LIN {X -0.022,Y -255.168,Z 987.708,A 0.000,B 0.000,C 90.000,E1 307.443} C_DIS
LIN {X -0.119,Y -266.430,Z 987.696,A 0.000,B 0.000,C 90.000,E1 305.311} C_DIS
LIN {X 0.015,Y -280.721,Z 987.682,A 0.000,B 0.000,C 90.000,E1 302.832} C_DIS
LIN {X -0.071,Y -295.961,Z 987.669,A 0.000,B 0.000,C 90.000,E1 300.463} C_DIS
LIN {X 0.194,Y -314.730,Z 987.654,A 0.000,B 0.000,C 90.000,E1 297.769} C_DIS
LIN {X -0.075,Y -330.365,Z 987.644,A 0.000,B 0.000,C 90.000,E1 295.899} C_DIS
LIN {X -0.054,Y -352.007,Z 987.631,A 0.000,B 0.000,C 90.000,E1 293.567} C_DIS
LIN {X 0.003,Y -370.661,Z 987.621,A 0.000,B 0.000,C 90.000,E1 291.716} C_DIS
LIN {X -0.030,Y -387.055,Z 987.612,A 0.000,B 0.000,C 90.000,E1 290.174} C_DIS
LIN {X 0.079,Y -397.816,Z 987.606,A 0.000,B 0.000,C 90.000,E1 289.141} C_DIS
LIN {X 0.039,Y -408.356,Z 987.601,A 0.000,B 0.000,C 90.000,E1 288.127} C_DIS
LIN {X -0.163,Y -415.784,Z 987.597,A 0.000,B 0.000,C 90.000,E1 287.402} C_DIS
LIN {X 0.003,Y -425.654,Z 987.591,A 0.000,B 0.000,C 90.000,E1 286.315} C_DIS
LIN {X -0.019,Y -435.159,Z 987.585,A 0.000,B 0.000,C 90.000,E1 285.245} C_DIS
LIN {X 0.027,Y -444.217,Z 987.579,A 0.000,B 0.000,C 90.000,E1 284.175} C_DIS
LIN {X 0.074,Y -452.686,Z 987.573,A 0.000,B 0.000,C 90.000,E1 283.119} C_DIS
LIN {X -0.041,Y -458.562,Z 987.569,A 0.000,B 0.000,C 90.000,E1 282.355} C_DIS
LIN {X 0.178,Y -465.822,Z 987.563,A 0.000,B 0.000,C 90.000,E1 281.299} C_DIS
LIN {X 0.080,Y -470.862,Z 987.559,A 0.000,B 0.000,C 90.000,E1 280.546} C_DIS
LIN {X 0.034,Y -475.472,Z 987.554,A 0.000,B 0.000,C 90.000,E1 279.792} C_DIS
LIN {X 0.101,Y -479.412,Z 987.550,A 0.000,B 0.000,C 90.000,E1 279.029} C_DIS
LIN {X 0.128,Y -482.743,Z 987.546,A 0.000,B 0.000,C 90.000,E1 278.276} C_DIS
LIN {X 0.117,Y -485.467,Z 987.542,A 0.000,B 0.000,C 90.000,E1 277.530} C_DIS
LIN {X -0.179,Y -486.911,Z 987.539,A 0.000,B 0.000,C 90.000,E1 277.068} C_DIS
LIN {X 0.019,Y -488.089,Z 987.536,A 0.000,B 0.000,C 90.000,E1 276.549} C_DIS
LIN {X -0.260,Y -489.035,Z 987.534,A 0.000,B 0.000,C 90.000,E1 276.087} C_DIS
LIN {X -0.046,Y -489.695,Z 987.531,A 0.000,B 0.000,C 90.000,E1 275.568} C_DIS
LIN {X 0.171,Y -489.938,Z 987.528,A 0.000,B 0.000,C 90.000,E1 275.049} C_DIS
LIN {X -0.097,Y -489.761,Z 987.525,A 0.000,B 0.000,C 90.000,E1 274.588} C_DIS
LIN {X 0.086,Y -489.164,Z 987.523,A 0.000,B 0.000,C 90.000,E1 274.073} C_DIS
LIN {X -0.183,Y -488.056,Z 987.520,A 0.000,B 0.000,C 90.000,E1 273.612} C_DIS
LIN {X 0.027,Y -486.383,Z 987.517,A 0.000,B 0.000,C 90.000,E1 273.094} C_DIS
LIN {X 0.204,Y -484.065,Z 987.514,A 0.000,B 0.000,C 90.000,E1 272.579} C_DIS
LIN {X 0.043,Y -482.670,Z 987.513,A 0.000,B 0.000,C 90.000,E1 272.350} C_DIS
LIN {X 0.200,Y -479.159,Z 987.510,A 0.000,B 0.000,C 90.000,E1 271.835} C_DIS
LIN {X 0.049,Y -477.109,Z 987.509,A 0.000,B 0.000,C 90.000,E1 271.604} C_DIS
LIN {X 0.175,Y -472.171,Z 987.506,A 0.000,B 0.000,C 90.000,E1 271.088} C_DIS
LIN {X -0.020,Y -466.295,Z 987.503,A 0.000,B 0.000,C 90.000,E1 270.630} C_DIS
LIN {X -0.205,Y -460.113,Z 987.501,A 0.000,B 0.000,C 90.000,E1 270.229} C_DIS
LIN {X 0.033,Y -453.441,Z 987.499,A 0.000,B 0.000,C 90.000,E1 269.828} C_DIS
LIN {X -0.169,Y -446.515,Z 987.497,A 0.000,B 0.000,C 90.000,E1 269.542} C_DIS
LIN {X 0.037,Y -439.143,Z 987.496,A 0.000,B 0.000,C 90.000,E1 269.255} C_DIS
LIN {X -0.206,Y -431.354,Z 987.495,A 0.000,B 0.000,C 90.000,E1 269.083} C_DIS
LIN {X -0.075,Y -423.163,Z 987.494,A 0.000,B 0.000,C 90.000,E1 268.912} C_DIS
LIN {X -0.046,Y -415.029,Z 987.493,A 0.000,B 0.000,C 90.000,E1 268.797} C_DIS
LIN {X -0.113,Y -407.726,Z 987.493,A 0.000,B 0.000,C 90.000,E1 268.740} C_DIS
LIN {X 0.081,Y -401.384,Z 987.493,A 0.000,B 0.000,C 90.000,E1 268.682} C_DIS
LIN {X 0.014,Y -181.252,Z 987.493,A 0.000,B 0.000,C 90.000,E1 268.682} C_DIS
LIN {X -0.081,Y -180.902,Z 987.474,A 0.000,B 0.000,C 90.000,E1 265.298} C_DIS
LIN {X 0.048,Y -180.232,Z 987.464,A 0.000,B 0.000,C 90.000,E1 263.571} C_DIS
LIN {X 0.065,Y -178.715,Z 987.441,A 0.000,B 0.000,C 90.000,E1 259.342} C_DIS
LIN {X -0.043,Y -175.763,Z 987.413,A 0.000,B 0.000,C 90.000,E1 254.283} C_DIS
LIN {X 0.007,Y -171.947,Z 987.384,A 0.000,B 0.000,C 90.000,E1 249.135} C_DIS
LIN {X -0.017,Y -171.334,Z 987.379,A 0.000,B 0.000,C 90.000,E1 248.284} C_DIS
LIN {X 0.035,Y -167.589,Z 987.355,A 0.000,B 0.000,C 90.000,E1 243.948} C_DIS
LIN {X -0.025,Y -166.226,Z 987.346,A 0.000,B 0.000,C 90.000,E1 242.231} C_DIS
LIN {X -0.037,Y -162.987,Z 987.326,A 0.000,B 0.000,C 90.000,E1 238.742} C_DIS
LIN {X 0.011,Y -160.904,Z 987.312,A 0.000,B 0.000,C 90.000,E1 236.087} C_DIS
LIN {X -0.012,Y -157.670,Z 987.292,A 0.000,B 0.000,C 90.000,E1 232.557} C_DIS
LIN {X -0.074,Y -155.709,Z 987.277,A 0.000,B 0.000,C 90.000,E1 229.908} C_DIS
LIN {X -0.019,Y -151.970,Z 987.252,A 0.000,B 0.000,C 90.000,E1 225.405} C_DIS
LIN {X -0.002,Y -150.213,Z 987.237,A 0.000,B 0.000,C 90.000,E1 222.690} C_DIS
LIN {X -0.078,Y -146.979,Z 987.212,A 0.000,B 0.000,C 90.000,E1 218.177} C_DIS
LIN {X 0.031,Y -145.565,Z 987.197,A 0.000,B 0.000,C 90.000,E1 215.391} C_DIS
LIN {X 0.030,Y -142.956,Z 987.171,A 0.000,B 0.000,C 90.000,E1 210.797} C_DIS
LIN {X -0.040,Y -141.582,Z 987.151,A 0.000,B 0.000,C 90.000,E1 207.129} C_DIS
LIN {X 0.008,Y -139.416,Z 987.115,A 0.000,B 0.000,C 90.000,E1 200.610} C_DIS
LIN {X 0.060,Y -139.142,Z 987.104,A 0.000,B 0.000,C 90.000,E1 198.725} C_DIS
LIN {X -0.049,Y -138.347,Z 987.057,A 0.000,B 0.000,C 90.000,E1 190.366} C_DIS
LIN {X -0.064,Y -139.491,Z 987.006,A 0.000,B 0.000,C 90.000,E1 181.031} C_DIS
LIN {X 0.016,Y -141.101,Z 986.975,A 0.000,B 0.000,C 90.000,E1 175.412} C_DIS
LIN {X -0.030,Y -142.479,Z 986.959,A 0.000,B 0.000,C 90.000,E1 172.648} C_DIS
LIN {X 0.058,Y -144.728,Z 986.933,A 0.000,B 0.000,C 90.000,E1 167.993} C_DIS
LIN {X 0.010,Y -147.332,Z 986.913,A 0.000,B 0.000,C 90.000,E1 164.338} C_DIS
LIN {X 0.075,Y -150.655,Z 986.888,A 0.000,B 0.000,C 90.000,E1 159.752} C_DIS
LIN {X -0.044,Y -154.132,Z 986.868,A 0.000,B 0.000,C 90.000,E1 156.177} C_DIS
LIN {X 0.019,Y -157.561,Z 986.848,A 0.000,B 0.000,C 90.000,E1 152.564} C_DIS
LIN {X 0.043,Y -161.803,Z 986.828,A 0.000,B 0.000,C 90.000,E1 148.997} C_DIS
LIN {X 0.063,Y -165.994,Z 986.808,A 0.000,B 0.000,C 90.000,E1 145.468} C_DIS
LIN {X 0.056,Y -170.992,Z 986.789,A 0.000,B 0.000,C 90.000,E1 141.984} C_DIS
LIN {X -0.028,Y -175.861,Z 986.770,A 0.000,B 0.000,C 90.000,E1 138.566} C_DIS
LIN {X -0.035,Y -181.466,Z 986.751,A 0.000,B 0.000,C 90.000,E1 135.162} C_DIS
LIN {X 0.102,Y -186.978,Z 986.732,A 0.000,B 0.000,C 90.000,E1 131.757} C_DIS
LIN {X 0.104,Y -190.093,Z 986.723,A 0.000,B 0.000,C 90.000,E1 130.092} C_DIS
LIN {X -0.044,Y -195.659,Z 986.705,A 0.000,B 0.000,C 90.000,E1 126.950} C_DIS
LIN {X -0.102,Y -299.362,Z 986.705,A 0.000,B 0.000,C 90.000,E1 126.950} C_DIS
LIN {X 0.011,Y -303.410,Z 986.705,A 0.000,B 0.000,C 90.000,E1 126.824} C_DIS
LIN {X -0.025,Y -306.209,Z 986.704,A 0.000,B 0.000,C 90.000,E1 126.664} C_DIS
LIN {X -0.013,Y -309.928,Z 986.702,A 0.000,B 0.000,C 90.000,E1 126.297} C_DIS
LIN {X 0.089,Y -313.456,Z 986.699,A 0.000,B 0.000,C 90.000,E1 125.724} C_DIS
LIN {X 0.133,Y -314.911,Z 986.697,A 0.000,B 0.000,C 90.000,E1 125.391} C_DIS
LIN {X 0.098,Y -320.171,Z 986.688,A 0.000,B 0.000,C 90.000,E1 123.785} C_DIS
LIN {X 0.110,Y -330.327,Z 986.672,A 0.000,B 0.000,C 90.000,E1 120.924} C_DIS
LIN {X -0.110,Y -341.814,Z 986.656,A 0.000,B 0.000,C 90.000,E1 118.153} C_DIS
LIN {X -0.180,Y -354.728,Z 986.641,A 0.000,B 0.000,C 90.000,E1 115.412} C_DIS
LIN {X -0.111,Y -367.502,Z 986.628,A 0.000,B 0.000,C 90.000,E1 113.003} C_DIS
LIN {X 0.198,Y -381.586,Z 986.615,A 0.000,B 0.000,C 90.000,E1 110.610} C_DIS
LIN {X -0.115,Y -397.080,Z 986.602,A 0.000,B 0.000,C 90.000,E1 108.362} C_DIS
LIN {X 0.208,Y -414.096,Z 986.589,A 0.000,B 0.000,C 90.000,E1 106.079} C_DIS
LIN {X -0.084,Y -432.754,Z 986.577,A 0.000,B 0.000,C 90.000,E1 103.939} C_DIS
LIN {X 0.243,Y -452.686,Z 986.566,A 0.000,B 0.000,C 90.000,E1 101.827} C_DIS
LIN {X -0.051,Y -467.898,Z 986.558,A 0.000,B 0.000,C 90.000,E1 100.423} C_DIS
LIN {X -0.110,Y -469.778,Z 986.557,A 0.000,B 0.000,C 90.000,E1 100.197} C_DIS
LIN {X 0.204,Y -471.333,Z 986.555,A 0.000,B 0.000,C 90.000,E1 99.905} C_DIS
LIN {X 0.054,Y -472.498,Z 986.554,A 0.000,B 0.000,C 90.000,E1 99.670} C_DIS
LIN {X 0.159,Y -473.903,Z 986.551,A 0.000,B 0.000,C 90.000,E1 99.151} C_DIS
LIN {X -0.123,Y -474.283,Z 986.548,A 0.000,B 0.000,C 90.000,E1 98.681} C_DIS
LIN {X -0.001,Y -473.700,Z 986.545,A 0.000,B 0.000,C 90.000,E1 98.163} C_DIS
LIN {X 0.124,Y -472.065,Z 986.543,A 0.000,B 0.000,C 90.000,E1 97.644} C_DIS
LIN {X -0.017,Y -470.765,Z 986.541,A 0.000,B 0.000,C 90.000,E1 97.409} C_DIS
LIN {X 0.045,Y -458.859,Z 986.531,A 0.000,B 0.000,C 90.000,E1 95.625} C_DIS
LIN {X 0.084,Y -448.473,Z 986.523,A 0.000,B 0.000,C 90.000,E1 94.073} C_DIS
LIN {X 0.039,Y -428.315,Z 986.505,A 0.000,B 0.000,C 90.000,E1 90.917} C_DIS
LIN {X 0.135,Y -410.281,Z 986.487,A 0.000,B 0.000,C 90.000,E1 87.650} C_DIS
LIN {X 0.151,Y -401.338,Z 986.478,A 0.000,B 0.000,C 90.000,E1 85.988} C_DIS
LIN {X 0.077,Y -390.622,Z 986.467,A 0.000,B 0.000,C 90.000,E1 84.033} C_DIS
LIN {X -0.147,Y -381.201,Z 986.457,A 0.000,B 0.000,C 90.000,E1 82.356} C_DIS
LIN {X -0.157,Y -371.588,Z 986.448,A 0.000,B 0.000,C 90.000,E1 80.622} C_DIS
LIN {X 0.138,Y -361.640,Z 986.438,A 0.000,B 0.000,C 90.000,E1 78.814} C_DIS
LIN {X -0.080,Y -349.979,Z 986.426,A 0.000,B 0.000,C 90.000,E1 76.756} C_DIS
LIN {X -0.009,Y -333.809,Z 986.409,A 0.000,B 0.000,C 90.000,E1 73.685} C_DIS
LIN {X 0.048,Y -321.441,Z 986.395,A 0.000,B 0.000,C 90.000,E1 71.167} C_DIS
LIN {X 0.113,Y -309.290,Z 986.381,A 0.000,B 0.000,C 90.000,E1 68.592} C_DIS
LIN {X 0.108,Y -298.848,Z 986.368,A 0.000,B 0.000,C 90.000,E1 66.305} C_DIS
LIN {X -0.141,Y -288.609,Z 986.356,A 0.000,B 0.000,C 90.000,E1 64.024} C_DIS
LIN {X -0.095,Y -278.482,Z 986.342,A 0.000,B 0.000,C 90.000,E1 61.641} C_DIS
LIN {X -0.077,Y -267.084,Z 986.327,A 0.000,B 0.000,C 90.000,E1 58.869} C_DIS
LIN {X 0.068,Y -255.979,Z 986.311,A 0.000,B 0.000,C 90.000,E1 56.008} C_DIS
LIN {X 0.017,Y -244.066,Z 986.293,A 0.000,B 0.000,C 90.000,E1 52.763} C_DIS
LIN {X -0.111,Y -232.938,Z 986.275,A 0.000,B 0.000,C 90.000,E1 49.461} C_DIS
LIN {X -0.109,Y -222.406,Z 986.256,A 0.000,B 0.000,C 90.000,E1 46.053} C_DIS
LIN {X 0.013,Y -213.683,Z 986.239,A 0.000,B 0.000,C 90.000,E1 42.933} C_DIS
LIN {X -0.041,Y -205.517,Z 986.221,A 0.000,B 0.000,C 90.000,E1 39.806} C_DIS
LIN {X 0.044,Y -197.992,Z 986.203,A 0.000,B 0.000,C 90.000,E1 36.583} C_DIS
LIN {X -0.090,Y -191.173,Z 986.185,A 0.000,B 0.000,C 90.000,E1 33.372} C_DIS
LIN {X -0.015,Y -185.059,Z 986.167,A 0.000,B 0.000,C 90.000,E1 30.050} C_DIS
LIN {X 0.022,Y -179.703,Z 986.148,A 0.000,B 0.000,C 90.000,E1 26.693} C_DIS
LIN {X -0.059,Y -175.100,Z 986.130,A 0.000,B 0.000,C 90.000,E1 23.334} C_DIS
LIN {X 0.024,Y -171.216,Z 986.111,A 0.000,B 0.000,C 90.000,E1 19.885} C_DIS
LIN {X 0.065,Y -167.326,Z 986.087,A 0.000,B 0.000,C 90.000,E1 15.552} C_DIS
LIN {X -0.073,Y -164.550,Z 986.062,A 0.000,B 0.000,C 90.000,E1 11.243} C_DIS
LIN {X 0.074,Y -162.303,Z 986.028,A 0.000,B 0.000,C 90.000,E1 5.049} C_DIS
LIN {X 0.085,Y -163.439,Z 985.963,A 0.000,B 0.000,C 90.000,E1 353.337} C_DIS
LIN {X -0.039,Y -165.698,Z 985.939,A 0.000,B 0.000,C 90.000,E1 348.993} C_DIS
LIN {X -0.031,Y -169.051,Z 985.915,A 0.000,B 0.000,C 90.000,E1 344.629} C_DIS
LIN {X 0.024,Y -172.607,Z 985.895,A 0.000,B 0.000,C 90.000,E1 341.148} C_DIS
LIN {X 0.010,Y -176.936,Z 985.876,A 0.000,B 0.000,C 90.000,E1 337.720} C_DIS
LIN {X -0.022,Y -181.986,Z 985.857,A 0.000,B 0.000,C 90.000,E1 334.332} C_DIS
LIN {X -0.020,Y -187.852,Z 985.839,A 0.000,B 0.000,C 90.000,E1 330.973} C_DIS
LIN {X -0.022,Y -194.450,Z 985.820,A 0.000,B 0.000,C 90.000,E1 327.661} C_DIS
LIN {X -0.041,Y -201.567,Z 985.802,A 0.000,B 0.000,C 90.000,E1 324.402} C_DIS
LIN {X -0.081,Y -210.239,Z 985.782,A 0.000,B 0.000,C 90.000,E1 320.803} C_DIS
LIN {X -0.002,Y -218.406,Z 985.765,A 0.000,B 0.000,C 90.000,E1 317.634} C_DIS
LIN {X -0.117,Y -228.247,Z 985.745,A 0.000,B 0.000,C 90.000,E1 314.190} C_DIS
LIN {X 0.127,Y -233.159,Z 985.737,A 0.000,B 0.000,C 90.000,E1 312.609} C_DIS
LIN {X -0.054,Y -238.830,Z 985.729,A 0.000,B 0.000,C 90.000,E1 311.148} C_DIS
LIN {X 0.001,Y -248.341,Z 985.716,A 0.000,B 0.000,C 90.000,E1 308.910} C_DIS
LIN {X -0.069,Y -258.902,Z 985.704,A 0.000,B 0.000,C 90.000,E1 306.744} C_DIS
LIN {X -0.105,Y -274.483,Z 985.688,A 0.000,B 0.000,C 90.000,E1 303.913} C_DIS
LIN {X 0.035,Y -291.567,Z 985.673,A 0.000,B 0.000,C 90.000,E1 301.131} C_DIS
LIN {X -0.045,Y -312.262,Z 985.656,A 0.000,B 0.000,C 90.000,E1 298.153} C_DIS
LIN {X -0.056,Y -325.012,Z 985.647,A 0.000,B 0.000,C 90.000,E1 296.539} C_DIS
LIN {X -0.158,Y -338.453,Z 985.639,A 0.000,B 0.000,C 90.000,E1 295.027} C_DIS
LIN {X 0.030,Y -362.458,Z 985.625,A 0.000,B 0.000,C 90.000,E1 292.514} C_DIS
LIN {X 0.074,Y -381.416,Z 985.615,A 0.000,B 0.000,C 90.000,E1 290.684} C_DIS
LIN {X -0.190,Y -394.934,Z 985.608,A 0.000,B 0.000,C 90.000,E1 289.450} C_DIS
LIN {X -0.118,Y -405.542,Z 985.602,A 0.000,B 0.000,C 90.000,E1 288.417} C_DIS
LIN {X -0.099,Y -413.272,Z 985.598,A 0.000,B 0.000,C 90.000,E1 287.638} C_DIS
LIN {X 0.077,Y -423.265,Z 985.592,A 0.000,B 0.000,C 90.000,E1 286.551} C_DIS
LIN {X 0.038,Y -432.890,Z 985.586,A 0.000,B 0.000,C 90.000,E1 285.481} C_DIS
LIN {X 0.058,Y -442.054,Z 985.580,A 0.000,B 0.000,C 90.000,E1 284.411} C_DIS
LIN {X 0.079,Y -450.649,Z 985.574,A 0.000,B 0.000,C 90.000,E1 283.355} C_DIS
LIN {X -0.060,Y -456.684,Z 985.570,A 0.000,B 0.000,C 90.000,E1 282.591} C_DIS
LIN {X 0.139,Y -464.119,Z 985.564,A 0.000,B 0.000,C 90.000,E1 281.535} C_DIS
LIN {X 0.030,Y -469.311,Z 985.560,A 0.000,B 0.000,C 90.000,E1 280.782} C_DIS
LIN {X 0.049,Y -474.042,Z 985.556,A 0.000,B 0.000,C 90.000,E1 280.018} C_DIS
LIN {X 0.029,Y -478.260,Z 985.552,A 0.000,B 0.000,C 90.000,E1 279.265} C_DIS
LIN {X 0.043,Y -481.831,Z 985.547,A 0.000,B 0.000,C 90.000,E1 278.511} C_DIS
LIN {X 0.209,Y -483.843,Z 985.545,A 0.000,B 0.000,C 90.000,E1 277.992} C_DIS
LIN {X -0.096,Y -485.608,Z 985.542,A 0.000,B 0.000,C 90.000,E1 277.530} C_DIS
LIN {X 0.093,Y -487.073,Z 985.539,A 0.000,B 0.000,C 90.000,E1 277.011} C_DIS
LIN {X -0.137,Y -488.244,Z 985.536,A 0.000,B 0.000,C 90.000,E1 276.543} C_DIS
LIN {X 0.015,Y -489.163,Z 985.534,A 0.000,B 0.000,C 90.000,E1 276.030} C_DIS
LIN {X -0.258,Y -489.822,Z 985.531,A 0.000,B 0.000,C 90.000,E1 275.568} C_DIS
LIN {X -0.039,Y -490.047,Z 985.528,A 0.000,B 0.000,C 90.000,E1 275.049} C_DIS
LIN {X 0.182,Y -489.897,Z 985.525,A 0.000,B 0.000,C 90.000,E1 274.531} C_DIS
LIN {X -0.122,Y -489.246,Z 985.523,A 0.000,B 0.000,C 90.000,E1 274.073} C_DIS
LIN {X 0.096,Y -488.113,Z 985.520,A 0.000,B 0.000,C 90.000,E1 273.555} C_DIS
LIN {X -0.179,Y -486.409,Z 985.517,A 0.000,B 0.000,C 90.000,E1 273.094} C_DIS
LIN {X -0.002,Y -484.065,Z 985.514,A 0.000,B 0.000,C 90.000,E1 272.579} C_DIS
LIN {X 0.163,Y -481.013,Z 985.512,A 0.000,B 0.000,C 90.000,E1 272.064} C_DIS
LIN {X -0.153,Y -477.050,Z 985.509,A 0.000,B 0.000,C 90.000,E1 271.604} C_DIS
LIN {X -0.025,Y -472.077,Z 985.506,A 0.000,B 0.000,C 90.000,E1 271.088} C_DIS
LIN {X -0.190,Y -466.220,Z 985.503,A 0.000,B 0.000,C 90.000,E1 270.630} C_DIS
LIN {X 0.122,Y -460.077,Z 985.501,A 0.000,B 0.000,C 90.000,E1 270.172} C_DIS
LIN {X -0.060,Y -453.504,Z 985.499,A 0.000,B 0.000,C 90.000,E1 269.828} C_DIS
LIN {X 0.163,Y -446.479,Z 985.497,A 0.000,B 0.000,C 90.000,E1 269.484} C_DIS
LIN {X -0.043,Y -439.233,Z 985.496,A 0.000,B 0.000,C 90.000,E1 269.255} C_DIS
LIN {X 0.151,Y -431.557,Z 985.495,A 0.000,B 0.000,C 90.000,E1 269.026} C_DIS
LIN {X -0.183,Y -423.307,Z 985.494,A 0.000,B 0.000,C 90.000,E1 268.912} C_DIS
LIN {X -0.176,Y -415.017,Z 985.493,A 0.000,B 0.000,C 90.000,E1 268.797} C_DIS
LIN {X 0.164,Y -407.332,Z 985.493,A 0.000,B 0.000,C 90.000,E1 268.682} C_DIS
LIN {X -0.046,Y -400.680,Z 985.493,A 0.000,B 0.000,C 90.000,E1 268.682} C_DIS
LIN {X -0.043,Y -181.248,Z 985.493,A 0.000,B 0.000,C 90.000,E1 268.682} C_DIS
LIN {X 0.045,Y -180.901,Z 985.474,A 0.000,B 0.000,C 90.000,E1 265.241} C_DIS
LIN {X -0.006,Y -180.224,Z 985.464,A 0.000,B 0.000,C 90.000,E1 263.571} C_DIS
LIN {X -0.053,Y -179.039,Z 985.445,A 0.000,B 0.000,C 90.000,E1 260.208} C_DIS
LIN {X 0.010,Y -178.704,Z 985.441,A 0.000,B 0.000,C 90.000,E1 259.342} C_DIS
LIN {X -0.049,Y -175.754,Z 985.413,A 0.000,B 0.000,C 90.000,E1 254.267} C_DIS
LIN {X -0.046,Y -171.936,Z 985.384,A 0.000,B 0.000,C 90.000,E1 249.135} C_DIS
LIN {X -0.070,Y -171.318,Z 985.379,A 0.000,B 0.000,C 90.000,E1 248.284} C_DIS
LIN {X -0.017,Y -167.576,Z 985.355,A 0.000,B 0.000,C 90.000,E1 243.948} C_DIS
LIN {X -0.078,Y -166.208,Z 985.346,A 0.000,B 0.000,C 90.000,E1 242.231} C_DIS
LIN {X -0.088,Y -162.973,Z 985.326,A 0.000,B 0.000,C 90.000,E1 238.742} C_DIS
LIN {X -0.040,Y -160.886,Z 985.312,A 0.000,B 0.000,C 90.000,E1 236.087} C_DIS
LIN {X -0.062,Y -157.655,Z 985.292,A 0.000,B 0.000,C 90.000,E1 232.557} C_DIS
LIN {X -0.005,Y -155.693,Z 985.277,A 0.000,B 0.000,C 90.000,E1 229.865} C_DIS
LIN {X -0.068,Y -151.958,Z 985.252,A 0.000,B 0.000,C 90.000,E1 225.405} C_DIS
LIN {X -0.051,Y -150.198,Z 985.237,A 0.000,B 0.000,C 90.000,E1 222.690} C_DIS
LIN {X 0.080,Y -146.968,Z 985.212,A 0.000,B 0.000,C 90.000,E1 218.096} C_DIS
LIN {X -0.017,Y -145.555,Z 985.197,A 0.000,B 0.000,C 90.000,E1 215.391} C_DIS
LIN {X -0.017,Y -142.947,Z 985.171,A 0.000,B 0.000,C 90.000,E1 210.797} C_DIS
LIN {X 0.039,Y -141.573,Z 985.151,A 0.000,B 0.000,C 90.000,E1 207.078} C_DIS
LIN {X -0.039,Y -139.413,Z 985.114,A 0.000,B 0.000,C 90.000,E1 200.610} C_DIS
LIN {X 0.013,Y -139.137,Z 985.104,A 0.000,B 0.000,C 90.000,E1 198.725} C_DIS
LIN {X 0.041,Y -138.349,Z 985.057,A 0.000,B 0.000,C 90.000,E1 190.310} C_DIS
LIN {X 0.028,Y -139.494,Z 985.005,A 0.000,B 0.000,C 90.000,E1 180.974} C_DIS
LIN {X -0.031,Y -141.109,Z 984.974,A 0.000,B 0.000,C 90.000,E1 175.412} C_DIS
LIN {X 0.063,Y -142.489,Z 984.959,A 0.000,B 0.000,C 90.000,E1 172.591} C_DIS
LIN {X 0.011,Y -144.739,Z 984.933,A 0.000,B 0.000,C 90.000,E1 167.993} C_DIS
LIN {X -0.040,Y -147.346,Z 984.913,A 0.000,B 0.000,C 90.000,E1 164.338} C_DIS
LIN {X 0.025,Y -150.671,Z 984.888,A 0.000,B 0.000,C 90.000,E1 159.752} C_DIS
LIN {X -0.094,Y -154.150,Z 984.867,A 0.000,B 0.000,C 90.000,E1 156.177} C_DIS
LIN {X 0.041,Y -157.580,Z 984.848,A 0.000,B 0.000,C 90.000,E1 152.538} C_DIS
LIN {X -0.008,Y -161.827,Z 984.828,A 0.000,B 0.000,C 90.000,E1 148.997} C_DIS
LIN {X 0.011,Y -166.018,Z 984.808,A 0.000,B 0.000,C 90.000,E1 145.468} C_DIS
LIN {X 0.003,Y -171.018,Z 984.789,A 0.000,B 0.000,C 90.000,E1 141.984} C_DIS
LIN {X 0.034,Y -175.889,Z 984.770,A 0.000,B 0.000,C 90.000,E1 138.528} C_DIS
LIN {X -0.090,Y -181.493,Z 984.751,A 0.000,B 0.000,C 90.000,E1 135.162} C_DIS
LIN {X 0.046,Y -187.009,Z 984.732,A 0.000,B 0.000,C 90.000,E1 131.757} C_DIS
LIN {X 0.047,Y -190.126,Z 984.723,A 0.000,B 0.000,C 90.000,E1 130.092} C_DIS
LIN {X 0.069,Y -195.598,Z 984.705,A 0.000,B 0.000,C 90.000,E1 126.950} C_DIS
LIN {X 0.070,Y -299.558,Z 984.705,A 0.000,B 0.000,C 90.000,E1 126.950} C_DIS
LIN {X -0.035,Y -300.837,Z 984.705,A 0.000,B 0.000,C 90.000,E1 126.950} C_DIS
LIN {X 0.104,Y -304.318,Z 984.704,A 0.000,B 0.000,C 90.000,E1 126.790} C_DIS
LIN {X -0.087,Y -307.597,Z 984.703,A 0.000,B 0.000,C 90.000,E1 126.583} C_DIS
LIN {X -0.046,Y -311.281,Z 984.701,A 0.000,B 0.000,C 90.000,E1 126.137} C_DIS
LIN {X 0.020,Y -313.164,Z 984.699,A 0.000,B 0.000,C 90.000,E1 125.804} C_DIS
LIN {X -0.168,Y -314.636,Z 984.697,A 0.000,B 0.000,C 90.000,E1 125.518} C_DIS
LIN {X -0.072,Y -317.828,Z 984.692,A 0.000,B 0.000,C 90.000,E1 124.532} C_DIS
LIN {X -0.033,Y -328.841,Z 984.674,A 0.000,B 0.000,C 90.000,E1 121.337} C_DIS
LIN {X 0.168,Y -340.141,Z 984.658,A 0.000,B 0.000,C 90.000,E1 118.487} C_DIS
LIN {X -0.098,Y -352.854,Z 984.643,A 0.000,B 0.000,C 90.000,E1 115.771} C_DIS
LIN {X 0.107,Y -365.434,Z 984.630,A 0.000,B 0.000,C 90.000,E1 113.334} C_DIS
LIN {X 0.163,Y -379.310,Z 984.617,A 0.000,B 0.000,C 90.000,E1 110.972} C_DIS
LIN {X -0.209,Y -394.581,Z 984.604,A 0.000,B 0.000,C 90.000,E1 108.725} C_DIS
LIN {X 0.046,Y -411.354,Z 984.591,A 0.000,B 0.000,C 90.000,E1 106.441} C_DIS
LIN {X 0.104,Y -429.752,Z 984.579,A 0.000,B 0.000,C 90.000,E1 104.245} C_DIS
LIN {X -0.093,Y -449.569,Z 984.568,A 0.000,B 0.000,C 90.000,E1 102.175} C_DIS
LIN {X -0.182,Y -467.385,Z 984.558,A 0.000,B 0.000,C 90.000,E1 100.489} C_DIS
LIN {X -0.188,Y -469.420,Z 984.557,A 0.000,B 0.000,C 90.000,E1 100.254} C_DIS
LIN {X -0.196,Y -470.965,Z 984.556,A 0.000,B 0.000,C 90.000,E1 100.018} C_DIS
LIN {X 0.121,Y -472.222,Z 984.554,A 0.000,B 0.000,C 90.000,E1 99.726} C_DIS
LIN {X -0.105,Y -473.145,Z 984.553,A 0.000,B 0.000,C 90.000,E1 99.500} C_DIS
LIN {X 0.082,Y -474.154,Z 984.550,A 0.000,B 0.000,C 90.000,E1 98.973} C_DIS
LIN {X 0.199,Y -474.181,Z 984.547,A 0.000,B 0.000,C 90.000,E1 98.454} C_DIS
LIN {X -0.144,Y -473.232,Z 984.544,A 0.000,B 0.000,C 90.000,E1 97.992} C_DIS
LIN {X 0.045,Y -471.147,Z 984.542,A 0.000,B 0.000,C 90.000,E1 97.466} C_DIS
LIN {X 0.041,Y -462.716,Z 984.534,A 0.000,B 0.000,C 90.000,E1 96.201} C_DIS
LIN {X 0.183,Y -452.477,Z 984.526,A 0.000,B 0.000,C 90.000,E1 94.645} C_DIS
LIN {X -0.074,Y -435.310,Z 984.511,A 0.000,B 0.000,C 90.000,E1 92.064} C_DIS
LIN {X -0.069,Y -421.057,Z 984.498,A 0.000,B 0.000,C 90.000,E1 89.656} C_DIS
LIN {X -0.093,Y -409.234,Z 984.486,A 0.000,B 0.000,C 90.000,E1 87.478} C_DIS
LIN {X -0.065,Y -400.243,Z 984.477,A 0.000,B 0.000,C 90.000,E1 85.812} C_DIS
LIN {X -0.146,Y -389.500,Z 984.466,A 0.000,B 0.000,C 90.000,E1 83.856} C_DIS
LIN {X -0.051,Y -380.055,Z 984.456,A 0.000,B 0.000,C 90.000,E1 82.129} C_DIS
LIN {X -0.029,Y -370.430,Z 984.447,A 0.000,B 0.000,C 90.000,E1 80.387} C_DIS
LIN {X -0.109,Y -360.441,Z 984.437,A 0.000,B 0.000,C 90.000,E1 78.634} C_DIS
LIN {X 0.001,Y -348.753,Z 984.425,A 0.000,B 0.000,C 90.000,E1 76.520} C_DIS
LIN {X 0.029,Y -332.658,Z 984.408,A 0.000,B 0.000,C 90.000,E1 73.449} C_DIS
LIN {X -0.099,Y -321.833,Z 984.396,A 0.000,B 0.000,C 90.000,E1 71.275} C_DIS
LIN {X -0.122,Y -309.702,Z 984.382,A 0.000,B 0.000,C 90.000,E1 68.720} C_DIS
LIN {X 0.013,Y -299.246,Z 984.369,A 0.000,B 0.000,C 90.000,E1 66.410} C_DIS
LIN {X 0.039,Y -288.996,Z 984.356,A 0.000,B 0.000,C 90.000,E1 64.076} C_DIS
LIN {X -0.035,Y -278.852,Z 984.343,A 0.000,B 0.000,C 90.000,E1 61.719} C_DIS
LIN {X -0.015,Y -267.423,Z 984.327,A 0.000,B 0.000,C 90.000,E1 58.948} C_DIS
LIN {X 0.132,Y -256.293,Z 984.312,A 0.000,B 0.000,C 90.000,E1 56.087} C_DIS
LIN {X 0.079,Y -244.370,Z 984.294,A 0.000,B 0.000,C 90.000,E1 52.844} C_DIS
LIN {X -0.042,Y -233.221,Z 984.275,A 0.000,B 0.000,C 90.000,E1 49.542} C_DIS
LIN {X -0.040,Y -222.704,Z 984.256,A 0.000,B 0.000,C 90.000,E1 46.134} C_DIS
LIN {X 0.135,Y -212.915,Z 984.237,A 0.000,B 0.000,C 90.000,E1 42.609} C_DIS
LIN {X 0.053,Y -204.817,Z 984.219,A 0.000,B 0.000,C 90.000,E1 39.483} C_DIS
LIN {X -0.007,Y -197.382,Z 984.202,A 0.000,B 0.000,C 90.000,E1 36.297} C_DIS
LIN {X 0.006,Y -190.635,Z 984.184,A 0.000,B 0.000,C 90.000,E1 33.038} C_DIS
LIN {X -0.028,Y -184.594,Z 984.165,A 0.000,B 0.000,C 90.000,E1 29.745} C_DIS
LIN {X 0.087,Y -179.312,Z 984.147,A 0.000,B 0.000,C 90.000,E1 26.360} C_DIS
LIN {X -0.012,Y -174.771,Z 984.128,A 0.000,B 0.000,C 90.000,E1 23.003} C_DIS
LIN {X -0.032,Y -170.109,Z 984.104,A 0.000,B 0.000,C 90.000,E1 18.725} C_DIS
LIN {X 0.084,Y -166.543,Z 984.080,A 0.000,B 0.000,C 90.000,E1 14.356} C_DIS
LIN {X -0.021,Y -163.675,Z 984.051,A 0.000,B 0.000,C 90.000,E1 9.151} C_DIS
LIN {X 0.013,Y -162.025,Z 984.002,A 0.000,B 0.000,C 90.000,E1 0.344} C_DIS
LIN {X 0.056,Y -163.877,Z 983.958,A 0.000,B 0.000,C 90.000,E1 352.470} C_DIS
LIN {X -0.028,Y -166.390,Z 983.934,A 0.000,B 0.000,C 90.000,E1 348.117} C_DIS
LIN {X -0.022,Y -169.160,Z 983.915,A 0.000,B 0.000,C 90.000,E1 344.629} C_DIS
LIN {X 0.036,Y -172.726,Z 983.895,A 0.000,B 0.000,C 90.000,E1 341.148} C_DIS
LIN {X 0.025,Y -177.081,Z 983.876,A 0.000,B 0.000,C 90.000,E1 337.720} C_DIS
LIN {X -0.003,Y -182.131,Z 983.857,A 0.000,B 0.000,C 90.000,E1 334.332} C_DIS
LIN {X 0.004,Y -188.007,Z 983.839,A 0.000,B 0.000,C 90.000,E1 330.973} C_DIS
LIN {X 0.007,Y -194.590,Z 983.820,A 0.000,B 0.000,C 90.000,E1 327.661} C_DIS
LIN {X -0.008,Y -201.675,Z 983.802,A 0.000,B 0.000,C 90.000,E1 324.402} C_DIS
LIN {X -0.044,Y -210.348,Z 983.782,A 0.000,B 0.000,C 90.000,E1 320.803} C_DIS
LIN {X 0.040,Y -218.497,Z 983.765,A 0.000,B 0.000,C 90.000,E1 317.634} C_DIS
LIN {X 0.001,Y -227.248,Z 983.747,A 0.000,B 0.000,C 90.000,E1 314.555} C_DIS
LIN {X -0.153,Y -233.388,Z 983.737,A 0.000,B 0.000,C 90.000,E1 312.690} C_DIS
LIN {X -0.001,Y -239.015,Z 983.729,A 0.000,B 0.000,C 90.000,E1 311.148} C_DIS
LIN {X 0.060,Y -248.472,Z 983.716,A 0.000,B 0.000,C 90.000,E1 308.910} C_DIS
LIN {X -0.005,Y -259.006,Z 983.704,A 0.000,B 0.000,C 90.000,E1 306.744} C_DIS
LIN {X -0.035,Y -274.547,Z 983.688,A 0.000,B 0.000,C 90.000,E1 303.913} C_DIS
LIN {X 0.111,Y -291.591,Z 983.673,A 0.000,B 0.000,C 90.000,E1 301.131} C_DIS
LIN {X 0.037,Y -312.261,Z 983.656,A 0.000,B 0.000,C 90.000,E1 298.153} C_DIS
LIN {X 0.029,Y -324.992,Z 983.647,A 0.000,B 0.000,C 90.000,E1 296.539} C_DIS
LIN {X -0.108,Y -338.453,Z 983.639,A 0.000,B 0.000,C 90.000,E1 295.027} C_DIS
LIN {X -0.129,Y -362.740,Z 983.625,A 0.000,B 0.000,C 90.000,E1 292.514} C_DIS
LIN {X -0.200,Y -384.545,Z 983.613,A 0.000,B 0.000,C 90.000,E1 290.429} C_DIS
LIN {X -0.037,Y -397.864,Z 983.606,A 0.000,B 0.000,C 90.000,E1 289.141} C_DIS
LIN {X -0.145,Y -408.390,Z 983.601,A 0.000,B 0.000,C 90.000,E1 288.127} C_DIS
LIN {X -0.043,Y -415.964,Z 983.596,A 0.000,B 0.000,C 90.000,E1 287.330} C_DIS
LIN {X -0.105,Y -425.980,Z 983.590,A 0.000,B 0.000,C 90.000,E1 286.260} C_DIS
LIN {X -0.167,Y -435.521,Z 983.584,A 0.000,B 0.000,C 90.000,E1 285.190} C_DIS
LIN {X -0.117,Y -444.502,Z 983.578,A 0.000,B 0.000,C 90.000,E1 284.120} C_DIS
LIN {X -0.068,Y -452.903,Z 983.573,A 0.000,B 0.000,C 90.000,E1 283.063} C_DIS
LIN {X 0.087,Y -460.662,Z 983.567,A 0.000,B 0.000,C 90.000,E1 282.007} C_DIS
LIN {X -0.123,Y -467.835,Z 983.561,A 0.000,B 0.000,C 90.000,E1 281.007} C_DIS
LIN {X 0.118,Y -474.259,Z 983.555,A 0.000,B 0.000,C 90.000,E1 279.962} C_DIS
LIN {X 0.102,Y -478.461,Z 983.551,A 0.000,B 0.000,C 90.000,E1 279.208} C_DIS
LIN {X 0.120,Y -482.009,Z 983.547,A 0.000,B 0.000,C 90.000,E1 278.454} C_DIS
LIN {X -0.191,Y -484.054,Z 983.544,A 0.000,B 0.000,C 90.000,E1 277.992} C_DIS
LIN {X 0.047,Y -485.820,Z 983.542,A 0.000,B 0.000,C 90.000,E1 277.466} C_DIS
LIN {X 0.234,Y -487.281,Z 983.539,A 0.000,B 0.000,C 90.000,E1 276.947} C_DIS
LIN {X -0.054,Y -488.437,Z 983.536,A 0.000,B 0.000,C 90.000,E1 276.486} C_DIS
LIN {X 0.152,Y -489.318,Z 983.533,A 0.000,B 0.000,C 90.000,E1 275.967} C_DIS
LIN {X -0.170,Y -489.925,Z 983.531,A 0.000,B 0.000,C 90.000,E1 275.511} C_DIS
LIN {X 0.050,Y -490.155,Z 983.528,A 0.000,B 0.000,C 90.000,E1 274.992} C_DIS
LIN {X -0.217,Y -489.956,Z 983.525,A 0.000,B 0.000,C 90.000,E1 274.531} C_DIS
LIN {X 0.002,Y -489.279,Z 983.522,A 0.000,B 0.000,C 90.000,E1 274.012} C_DIS
LIN {X 0.187,Y -488.100,Z 983.520,A 0.000,B 0.000,C 90.000,E1 273.498} C_DIS
LIN {X 0.243,Y -485.250,Z 983.515,A 0.000,B 0.000,C 90.000,E1 272.751} C_DIS
LIN {X -0.071,Y -482.501,Z 983.513,A 0.000,B 0.000,C 90.000,E1 272.293} C_DIS
LIN {X 0.101,Y -478.933,Z 983.510,A 0.000,B 0.000,C 90.000,E1 271.776} C_DIS
LIN {X 0.235,Y -474.418,Z 983.507,A 0.000,B 0.000,C 90.000,E1 271.260} C_DIS
LIN {X 0.007,Y -468.961,Z 983.504,A 0.000,B 0.000,C 90.000,E1 270.802} C_DIS
LIN {X 0.132,Y -462.975,Z 983.502,A 0.000,B 0.000,C 90.000,E1 270.344} C_DIS
LIN {X 0.227,Y -456.598,Z 983.500,A 0.000,B 0.000,C 90.000,E1 269.943} C_DIS
LIN {X -0.169,Y -449.888,Z 983.498,A 0.000,B 0.000,C 90.000,E1 269.656} C_DIS
LIN {X -0.134,Y -442.796,Z 983.496,A 0.000,B 0.000,C 90.000,E1 269.370} C_DIS
LIN {X -0.122,Y -435.264,Z 983.495,A 0.000,B 0.000,C 90.000,E1 269.141} C_DIS
LIN {X -0.166,Y -427.592,Z 983.494,A 0.000,B 0.000,C 90.000,E1 268.969} C_DIS
LIN {X 0.101,Y -419.318,Z 983.493,A 0.000,B 0.000,C 90.000,E1 268.797} C_DIS
LIN {X 0.017,Y -406.774,Z 983.493,A 0.000,B 0.000,C 90.000,E1 268.682} C_DIS
LIN {X -0.141,Y -401.554,Z 983.493,A 0.000,B 0.000,C 90.000,E1 268.682} C_DIS
LIN {X -0.085,Y -181.245,Z 983.493,A 0.000,B 0.000,C 90.000,E1 268.682} C_DIS
LIN {X -0.013,Y -180.900,Z 983.474,A 0.000,B 0.000,C 90.000,E1 265.241} C_DIS
LIN {X -0.063,Y -180.215,Z 983.464,A 0.000,B 0.000,C 90.000,E1 263.571} C_DIS
LIN {X 0.067,Y -179.034,Z 983.445,A 0.000,B 0.000,C 90.000,E1 260.151} C_DIS
LIN {X -0.047,Y -178.693,Z 983.441,A 0.000,B 0.000,C 90.000,E1 259.342} C_DIS
LIN {X 0.064,Y -175.741,Z 983.412,A 0.000,B 0.000,C 90.000,E1 254.212} C_DIS
LIN {X 0.059,Y -171.925,Z 983.384,A 0.000,B 0.000,C 90.000,E1 249.082} C_DIS
LIN {X 0.034,Y -171.300,Z 983.379,A 0.000,B 0.000,C 90.000,E1 248.230} C_DIS
LIN {X 0.079,Y -167.562,Z 983.355,A 0.000,B 0.000,C 90.000,E1 243.896} C_DIS
LIN {X 0.092,Y -166.188,Z 983.345,A 0.000,B 0.000,C 90.000,E1 242.153} C_DIS
LIN {X 0.082,Y -162.957,Z 983.326,A 0.000,B 0.000,C 90.000,E1 238.663} C_DIS
LIN {X -0.094,Y -160.866,Z 983.311,A 0.000,B 0.000,C 90.000,E1 236.087} C_DIS
LIN {X 0.010,Y -157.640,Z 983.292,A 0.000,B 0.000,C 90.000,E1 232.512} C_DIS
LIN {X 0.043,Y -155.677,Z 983.277,A 0.000,B 0.000,C 90.000,E1 229.828} C_DIS
LIN {X -0.011,Y -151.944,Z 983.252,A 0.000,B 0.000,C 90.000,E1 225.364} C_DIS
LIN {X -0.102,Y -150.182,Z 983.237,A 0.000,B 0.000,C 90.000,E1 222.690} C_DIS
LIN {X 0.029,Y -146.956,Z 983.212,A 0.000,B 0.000,C 90.000,E1 218.096} C_DIS
LIN {X -0.068,Y -145.544,Z 983.196,A 0.000,B 0.000,C 90.000,E1 215.391} C_DIS
LIN {X -0.067,Y -142.939,Z 983.171,A 0.000,B 0.000,C 90.000,E1 210.797} C_DIS
LIN {X -0.010,Y -141.563,Z 983.150,A 0.000,B 0.000,C 90.000,E1 207.078} C_DIS
LIN {X 0.043,Y -139.409,Z 983.114,A 0.000,B 0.000,C 90.000,E1 200.556} C_DIS
LIN {X -0.035,Y -139.131,Z 983.104,A 0.000,B 0.000,C 90.000,E1 198.725} C_DIS
LIN {X -0.008,Y -138.350,Z 983.057,A 0.000,B 0.000,C 90.000,E1 190.310} C_DIS
LIN {X -0.021,Y -139.497,Z 983.005,A 0.000,B 0.000,C 90.000,E1 180.974} C_DIS
LIN {X 0.060,Y -141.118,Z 982.974,A 0.000,B 0.000,C 90.000,E1 175.355} C_DIS
LIN {X 0.014,Y -142.497,Z 982.959,A 0.000,B 0.000,C 90.000,E1 172.591} C_DIS
LIN {X -0.040,Y -144.752,Z 982.933,A 0.000,B 0.000,C 90.000,E1 167.993} C_DIS
LIN {X 0.052,Y -147.361,Z 982.913,A 0.000,B 0.000,C 90.000,E1 164.283} C_DIS
LIN {X -0.026,Y -150.688,Z 982.887,A 0.000,B 0.000,C 90.000,E1 159.752} C_DIS
LIN {X 0.057,Y -154.168,Z 982.867,A 0.000,B 0.000,C 90.000,E1 156.102} C_DIS
LIN {X -0.013,Y -157.601,Z 982.847,A 0.000,B 0.000,C 90.000,E1 152.538} C_DIS
LIN {X -0.062,Y -161.851,Z 982.828,A 0.000,B 0.000,C 90.000,E1 148.997} C_DIS
LIN {X -0.044,Y -166.042,Z 982.808,A 0.000,B 0.000,C 90.000,E1 145.468} C_DIS
LIN {X -0.053,Y -171.045,Z 982.789,A 0.000,B 0.000,C 90.000,E1 141.984} C_DIS
LIN {X -0.023,Y -175.917,Z 982.770,A 0.000,B 0.000,C 90.000,E1 138.528} C_DIS
LIN {X -0.030,Y -180.155,Z 982.755,A 0.000,B 0.000,C 90.000,E1 135.972} C_DIS
LIN {X -0.061,Y -185.572,Z 982.737,A 0.000,B 0.000,C 90.000,E1 132.609} C_DIS
LIN {X -0.012,Y -190.161,Z 982.723,A 0.000,B 0.000,C 90.000,E1 130.092} C_DIS
LIN {X 0.044,Y -195.526,Z 982.706,A 0.000,B 0.000,C 90.000,E1 126.996} C_DIS
LIN {X 0.032,Y -299.076,Z 982.706,A 0.000,B 0.000,C 90.000,E1 126.996} C_DIS
LIN {X -0.075,Y -300.591,Z 982.705,A 0.000,B 0.000,C 90.000,E1 126.996} C_DIS
LIN {X 0.009,Y -305.071,Z 982.704,A 0.000,B 0.000,C 90.000,E1 126.790} C_DIS
LIN {X 0.125,Y -308.249,Z 982.703,A 0.000,B 0.000,C 90.000,E1 126.503} C_DIS
LIN {X 0.156,Y -311.941,Z 982.700,A 0.000,B 0.000,C 90.000,E1 126.011} C_DIS
LIN {X -0.059,Y -313.673,Z 982.698,A 0.000,B 0.000,C 90.000,E1 125.724} C_DIS
LIN {X -0.021,Y -315.030,Z 982.697,A 0.000,B 0.000,C 90.000,E1 125.391} C_DIS
LIN {X -0.065,Y -326.846,Z 982.677,A 0.000,B 0.000,C 90.000,E1 121.878} C_DIS
LIN {X 0.081,Y -337.890,Z 982.661,A 0.000,B 0.000,C 90.000,E1 119.027} C_DIS
LIN {X -0.085,Y -350.329,Z 982.646,A 0.000,B 0.000,C 90.000,E1 116.283} C_DIS
LIN {X -0.070,Y -364.276,Z 982.631,A 0.000,B 0.000,C 90.000,E1 113.567} C_DIS
LIN {X -0.195,Y -378.037,Z 982.618,A 0.000,B 0.000,C 90.000,E1 111.227} C_DIS
LIN {X -0.107,Y -393.183,Z 982.605,A 0.000,B 0.000,C 90.000,E1 108.906} C_DIS
LIN {X 0.117,Y -409.823,Z 982.592,A 0.000,B 0.000,C 90.000,E1 106.622} C_DIS
LIN {X 0.142,Y -428.076,Z 982.580,A 0.000,B 0.000,C 90.000,E1 104.426} C_DIS
LIN {X -0.149,Y -447.816,Z 982.569,A 0.000,B 0.000,C 90.000,E1 102.355} C_DIS
LIN {X 0.234,Y -468.045,Z 982.558,A 0.000,B 0.000,C 90.000,E1 100.366} C_DIS
LIN {X 0.096,Y -469.957,Z 982.556,A 0.000,B 0.000,C 90.000,E1 100.141} C_DIS
LIN {X 0.042,Y -471.407,Z 982.555,A 0.000,B 0.000,C 90.000,E1 99.905} C_DIS
LIN {X 0.217,Y -473.376,Z 982.552,A 0.000,B 0.000,C 90.000,E1 99.378} C_DIS
LIN {X -0.146,Y -474.222,Z 982.549,A 0.000,B 0.000,C 90.000,E1 98.916} C_DIS
LIN {X -0.026,Y -474.094,Z 982.547,A 0.000,B 0.000,C 90.000,E1 98.398} C_DIS
LIN {X 0.166,Y -472.978,Z 982.544,A 0.000,B 0.000,C 90.000,E1 97.871} C_DIS
LIN {X -0.037,Y -471.998,Z 982.542,A 0.000,B 0.000,C 90.000,E1 97.644} C_DIS
LIN {X -0.177,Y -470.677,Z 982.541,A 0.000,B 0.000,C 90.000,E1 97.409} C_DIS
LIN {X 0.158,Y -457.104,Z 982.530,A 0.000,B 0.000,C 90.000,E1 95.334} C_DIS
LIN {X -0.093,Y -444.996,Z 982.520,A 0.000,B 0.000,C 90.000,E1 93.555} C_DIS
LIN {X 0.027,Y -426.754,Z 982.504,A 0.000,B 0.000,C 90.000,E1 90.630} C_DIS
LIN {X -0.095,Y -411.750,Z 982.488,A 0.000,B 0.000,C 90.000,E1 87.936} C_DIS
LIN {X -0.043,Y -402.814,Z 982.479,A 0.000,B 0.000,C 90.000,E1 86.274} C_DIS
LIN {X -0.077,Y -392.130,Z 982.468,A 0.000,B 0.000,C 90.000,E1 84.318} C_DIS
LIN {X 0.096,Y -381.138,Z 982.457,A 0.000,B 0.000,C 90.000,E1 82.299} C_DIS
LIN {X 0.078,Y -371.577,Z 982.448,A 0.000,B 0.000,C 90.000,E1 80.566} C_DIS
LIN {X 0.010,Y -361.581,Z 982.438,A 0.000,B 0.000,C 90.000,E1 78.814} C_DIS
LIN {X 0.131,Y -349.875,Z 982.426,A 0.000,B 0.000,C 90.000,E1 76.700} C_DIS
LIN {X -0.137,Y -333.701,Z 982.409,A 0.000,B 0.000,C 90.000,E1 73.685} C_DIS
LIN {X 0.026,Y -321.318,Z 982.395,A 0.000,B 0.000,C 90.000,E1 71.148} C_DIS
LIN {X -0.010,Y -309.226,Z 982.381,A 0.000,B 0.000,C 90.000,E1 68.592} C_DIS
LIN {X -0.003,Y -297.311,Z 982.367,A 0.000,B 0.000,C 90.000,E1 65.973} C_DIS
LIN {X -0.017,Y -287.066,Z 982.354,A 0.000,B 0.000,C 90.000,E1 63.640} C_DIS
LIN {X -0.009,Y -276.910,Z 982.340,A 0.000,B 0.000,C 90.000,E1 61.257} C_DIS
LIN {X 0.101,Y -265.523,Z 982.325,A 0.000,B 0.000,C 90.000,E1 58.456} C_DIS
LIN {X 0.089,Y -253.117,Z 982.307,A 0.000,B 0.000,C 90.000,E1 55.261} C_DIS
LIN {X 0.093,Y -241.347,Z 982.289,A 0.000,B 0.000,C 90.000,E1 51.984} C_DIS
LIN {X 0.035,Y -230.403,Z 982.270,A 0.000,B 0.000,C 90.000,E1 48.647} C_DIS
LIN {X -0.054,Y -220.105,Z 982.251,A 0.000,B 0.000,C 90.000,E1 45.243} C_DIS
LIN {X -0.082,Y -210.543,Z 982.232,A 0.000,B 0.000,C 90.000,E1 41.757} C_DIS
LIN {X 0.099,Y -202.613,Z 982.214,A 0.000,B 0.000,C 90.000,E1 38.543} C_DIS
LIN {X -0.015,Y -195.408,Z 982.196,A 0.000,B 0.000,C 90.000,E1 35.358} C_DIS
LIN {X 0.000,Y -188.871,Z 982.178,A 0.000,B 0.000,C 90.000,E1 32.084} C_DIS
LIN {X 0.080,Y -183.068,Z 982.160,A 0.000,B 0.000,C 90.000,E1 28.743} C_DIS
LIN {X -0.012,Y -177.984,Z 982.141,A 0.000,B 0.000,C 90.000,E1 25.412} C_DIS
LIN {X -0.049,Y -173.696,Z 982.122,A 0.000,B 0.000,C 90.000,E1 22.025} C_DIS
LIN {X -0.065,Y -170.053,Z 982.103,A 0.000,B 0.000,C 90.000,E1 18.598} C_DIS
LIN {X 0.004,Y -166.527,Z 982.079,A 0.000,B 0.000,C 90.000,E1 14.245} C_DIS
LIN {X -0.067,Y -163.693,Z 982.050,A 0.000,B 0.000,C 90.000,E1 9.029} C_DIS
LIN {X 0.030,Y -164.396,Z 981.953,A 0.000,B 0.000,C 90.000,E1 351.602} C_DIS
LIN {X 0.024,Y -167.116,Z 981.929,A 0.000,B 0.000,C 90.000,E1 347.229} C_DIS
LIN {X 0.054,Y -170.106,Z 981.910,A 0.000,B 0.000,C 90.000,E1 343.740} C_DIS
LIN {X 0.023,Y -173.876,Z 981.891,A 0.000,B 0.000,C 90.000,E1 340.296} C_DIS
LIN {X 0.037,Y -178.423,Z 981.872,A 0.000,B 0.000,C 90.000,E1 336.869} C_DIS
LIN {X -0.054,Y -183.691,Z 981.853,A 0.000,B 0.000,C 90.000,E1 333.512} C_DIS
LIN {X 0.076,Y -189.740,Z 981.834,A 0.000,B 0.000,C 90.000,E1 330.127} C_DIS
LIN {X 0.059,Y -196.451,Z 981.816,A 0.000,B 0.000,C 90.000,E1 326.834} C_DIS
LIN {X -0.072,Y -203.680,Z 981.798,A 0.000,B 0.000,C 90.000,E1 323.623} C_DIS
LIN {X 0.076,Y -212.434,Z 981.778,A 0.000,B 0.000,C 90.000,E1 319.989} C_DIS
LIN {X -0.036,Y -221.815,Z 981.758,A 0.000,B 0.000,C 90.000,E1 316.500} C_DIS
LIN {X 0.078,Y -229.787,Z 981.743,A 0.000,B 0.000,C 90.000,E1 313.785} C_DIS
LIN {X -0.031,Y -236.310,Z 981.733,A 0.000,B 0.000,C 90.000,E1 311.919} C_DIS
LIN {X 0.133,Y -245.347,Z 981.720,A 0.000,B 0.000,C 90.000,E1 309.644} C_DIS
LIN {X -0.051,Y -253.721,Z 981.710,A 0.000,B 0.000,C 90.000,E1 307.855} C_DIS
LIN {X 0.082,Y -266.677,Z 981.696,A 0.000,B 0.000,C 90.000,E1 305.311} C_DIS
LIN {X -0.003,Y -280.872,Z 981.683,A 0.000,B 0.000,C 90.000,E1 302.880} C_DIS
LIN {X 0.160,Y -298.300,Z 981.668,A 0.000,B 0.000,C 90.000,E1 300.129} C_DIS
LIN {X 0.017,Y -314.697,Z 981.655,A 0.000,B 0.000,C 90.000,E1 297.847} C_DIS
LIN {X 0.114,Y -330.162,Z 981.644,A 0.000,B 0.000,C 90.000,E1 295.924} C_DIS
LIN {X -0.115,Y -354.004,Z 981.630,A 0.000,B 0.000,C 90.000,E1 293.387} C_DIS
LIN {X -0.039,Y -370.164,Z 981.621,A 0.000,B 0.000,C 90.000,E1 291.770} C_DIS
LIN {X 0.049,Y -386.583,Z 981.612,A 0.000,B 0.000,C 90.000,E1 290.194} C_DIS
LIN {X 0.198,Y -399.839,Z 981.605,A 0.000,B 0.000,C 90.000,E1 288.906} C_DIS
LIN {X 0.195,Y -410.276,Z 981.599,A 0.000,B 0.000,C 90.000,E1 287.873} C_DIS
LIN {X -0.031,Y -420.248,Z 981.594,A 0.000,B 0.000,C 90.000,E1 286.858} C_DIS
LIN {X -0.093,Y -430.052,Z 981.588,A 0.000,B 0.000,C 90.000,E1 285.788} C_DIS
LIN {X -0.105,Y -439.312,Z 981.582,A 0.000,B 0.000,C 90.000,E1 284.717} C_DIS
LIN {X -0.009,Y -448.034,Z 981.576,A 0.000,B 0.000,C 90.000,E1 283.647} C_DIS
LIN {X 0.086,Y -456.180,Z 981.570,A 0.000,B 0.000,C 90.000,E1 282.591} C_DIS
LIN {X -0.174,Y -463.694,Z 981.564,A 0.000,B 0.000,C 90.000,E1 281.591} C_DIS
LIN {X 0.015,Y -470.625,Z 981.559,A 0.000,B 0.000,C 90.000,E1 280.546} C_DIS
LIN {X -0.033,Y -475.292,Z 981.554,A 0.000,B 0.000,C 90.000,E1 279.792} C_DIS
LIN {X 0.033,Y -479.371,Z 981.550,A 0.000,B 0.000,C 90.000,E1 279.029} C_DIS
LIN {X 0.058,Y -482.821,Z 981.546,A 0.000,B 0.000,C 90.000,E1 278.276} C_DIS
LIN {X 0.047,Y -485.628,Z 981.542,A 0.000,B 0.000,C 90.000,E1 277.530} C_DIS
LIN {X -0.248,Y -487.198,Z 981.539,A 0.000,B 0.000,C 90.000,E1 277.068} C_DIS
LIN {X -0.049,Y -488.417,Z 981.536,A 0.000,B 0.000,C 90.000,E1 276.549} C_DIS
LIN {X 0.159,Y -489.339,Z 981.534,A 0.000,B 0.000,C 90.000,E1 276.030} C_DIS
LIN {X -0.112,Y -489.951,Z 981.531,A 0.000,B 0.000,C 90.000,E1 275.568} C_DIS
LIN {X 0.107,Y -490.237,Z 981.528,A 0.000,B 0.000,C 90.000,E1 275.049} C_DIS
LIN {X -0.160,Y -490.115,Z 981.525,A 0.000,B 0.000,C 90.000,E1 274.588} C_DIS
LIN {X 0.026,Y -489.518,Z 981.523,A 0.000,B 0.000,C 90.000,E1 274.073} C_DIS
LIN {X -0.242,Y -488.366,Z 981.520,A 0.000,B 0.000,C 90.000,E1 273.612} C_DIS
LIN {X -0.029,Y -486.709,Z 981.517,A 0.000,B 0.000,C 90.000,E1 273.094} C_DIS
LIN {X 0.149,Y -484.399,Z 981.514,A 0.000,B 0.000,C 90.000,E1 272.579} C_DIS
LIN {X -0.167,Y -481.408,Z 981.512,A 0.000,B 0.000,C 90.000,E1 272.121} C_DIS
LIN {X 0.000,Y -477.549,Z 981.509,A 0.000,B 0.000,C 90.000,E1 271.604} C_DIS
LIN {X 0.128,Y -472.646,Z 981.506,A 0.000,B 0.000,C 90.000,E1 271.088} C_DIS
LIN {X -0.088,Y -466.786,Z 981.503,A 0.000,B 0.000,C 90.000,E1 270.630} C_DIS
LIN {X 0.187,Y -460.670,Z 981.501,A 0.000,B 0.000,C 90.000,E1 270.172} C_DIS
LIN {X -0.047,Y -454.096,Z 981.499,A 0.000,B 0.000,C 90.000,E1 269.828} C_DIS
LIN {X 0.129,Y -447.070,Z 981.497,A 0.000,B 0.000,C 90.000,E1 269.484} C_DIS
LIN {X -0.122,Y -439.694,Z 981.496,A 0.000,B 0.000,C 90.000,E1 269.255} C_DIS
LIN {X 0.059,Y -432.245,Z 981.495,A 0.000,B 0.000,C 90.000,E1 269.026} C_DIS
LIN {X 0.150,Y -424.484,Z 981.494,A 0.000,B 0.000,C 90.000,E1 268.854} C_DIS
LIN {X 0.082,Y -416.183,Z 981.493,A 0.000,B 0.000,C 90.000,E1 268.740} C_DIS
LIN {X -0.189,Y -404.862,Z 981.493,A 0.000,B 0.000,C 90.000,E1 268.682} C_DIS
LIN {X 0.156,Y -402.119,Z 981.492,A 0.000,B 0.000,C 90.000,E1 268.625} C_DIS
LIN {X 0.045,Y -181.241,Z 981.492,A 0.000,B 0.000,C 90.000,E1 268.625} C_DIS
LIN {X -0.068,Y -180.897,Z 981.473,A 0.000,B 0.000,C 90.000,E1 265.241} C_DIS
LIN {X -0.044,Y -179.848,Z 981.459,A 0.000,B 0.000,C 90.000,E1 262.704} C_DIS
LIN {X 0.013,Y -179.030,Z 981.445,A 0.000,B 0.000,C 90.000,E1 260.151} C_DIS
LIN {X 0.074,Y -178.681,Z 981.441,A 0.000,B 0.000,C 90.000,E1 259.285} C_DIS
LIN {X 0.011,Y -175.730,Z 981.412,A 0.000,B 0.000,C 90.000,E1 254.212} C_DIS
LIN {X 0.006,Y -171.916,Z 981.384,A 0.000,B 0.000,C 90.000,E1 249.082} C_DIS
LIN {X -0.019,Y -171.283,Z 981.379,A 0.000,B 0.000,C 90.000,E1 248.230} C_DIS
LIN {X 0.027,Y -167.549,Z 981.355,A 0.000,B 0.000,C 90.000,E1 243.896} C_DIS
LIN {X 0.041,Y -166.170,Z 981.345,A 0.000,B 0.000,C 90.000,E1 242.153} C_DIS
LIN {X 0.031,Y -162.943,Z 981.326,A 0.000,B 0.000,C 90.000,E1 238.663} C_DIS
LIN {X 0.008,Y -161.613,Z 981.316,A 0.000,B 0.000,C 90.000,E1 236.914} C_DIS
LIN {X -0.016,Y -159.140,Z 981.302,A 0.000,B 0.000,C 90.000,E1 234.276} C_DIS
LIN {X -0.006,Y -155.661,Z 981.277,A 0.000,B 0.000,C 90.000,E1 229.828} C_DIS
LIN {X 0.046,Y -151.931,Z 981.252,A 0.000,B 0.000,C 90.000,E1 225.324} C_DIS
LIN {X 0.061,Y -150.167,Z 981.237,A 0.000,B 0.000,C 90.000,E1 222.609} C_DIS
LIN {X -0.019,Y -146.945,Z 981.212,A 0.000,B 0.000,C 90.000,E1 218.096} C_DIS
LIN {X -0.031,Y -145.533,Z 981.196,A 0.000,B 0.000,C 90.000,E1 215.358} C_DIS
LIN {X 0.008,Y -142.930,Z 981.171,A 0.000,B 0.000,C 90.000,E1 210.747} C_DIS
LIN {X 0.008,Y -141.554,Z 981.150,A 0.000,B 0.000,C 90.000,E1 207.052} C_DIS
LIN {X -0.003,Y -139.407,Z 981.114,A 0.000,B 0.000,C 90.000,E1 200.556} C_DIS
LIN {X 0.050,Y -139.125,Z 981.104,A 0.000,B 0.000,C 90.000,E1 198.671} C_DIS
LIN {X -0.055,Y -138.351,Z 981.057,A 0.000,B 0.000,C 90.000,E1 190.310} C_DIS
LIN {X -0.067,Y -139.500,Z 981.005,A 0.000,B 0.000,C 90.000,E1 180.974} C_DIS
LIN {X 0.013,Y -141.125,Z 980.974,A 0.000,B 0.000,C 90.000,E1 175.355} C_DIS
LIN {X -0.033,Y -142.506,Z 980.959,A 0.000,B 0.000,C 90.000,E1 172.591} C_DIS
LIN {X 0.054,Y -144.763,Z 980.933,A 0.000,B 0.000,C 90.000,E1 167.937} C_DIS
LIN {X 0.003,Y -147.374,Z 980.913,A 0.000,B 0.000,C 90.000,E1 164.283} C_DIS
LIN {X 0.067,Y -150.703,Z 980.887,A 0.000,B 0.000,C 90.000,E1 159.699} C_DIS
LIN {X 0.007,Y -154.184,Z 980.867,A 0.000,B 0.000,C 90.000,E1 156.102} C_DIS
LIN {X 0.078,Y -157.620,Z 980.847,A 0.000,B 0.000,C 90.000,E1 152.487} C_DIS
LIN {X 0.026,Y -161.875,Z 980.828,A 0.000,B 0.000,C 90.000,E1 148.948} C_DIS
LIN {X -0.002,Y -166.066,Z 980.808,A 0.000,B 0.000,C 90.000,E1 145.435} C_DIS
LIN {X -0.001,Y -171.072,Z 980.789,A 0.000,B 0.000,C 90.000,E1 141.949} C_DIS
LIN {X 0.055,Y -175.944,Z 980.769,A 0.000,B 0.000,C 90.000,E1 138.485} C_DIS
LIN {X -0.085,Y -180.185,Z 980.755,A 0.000,B 0.000,C 90.000,E1 135.972} C_DIS
LIN {X -0.117,Y -185.602,Z 980.737,A 0.000,B 0.000,C 90.000,E1 132.609} C_DIS
LIN {X -0.068,Y -190.195,Z 980.723,A 0.000,B 0.000,C 90.000,E1 130.092} C_DIS
LIN {X 0.043,Y -195.464,Z 980.706,A 0.000,B 0.000,C 90.000,E1 127.030} C_DIS
LIN {X 0.019,Y -299.210,Z 980.706,A 0.000,B 0.000,C 90.000,E1 127.030} C_DIS
LIN {X -0.027,Y -299.941,Z 980.706,A 0.000,B 0.000,C 90.000,E1 127.030} C_DIS
LIN {X -0.080,Y -305.686,Z 980.704,A 0.000,B 0.000,C 90.000,E1 126.790} C_DIS
LIN {X -0.002,Y -308.667,Z 980.703,A 0.000,B 0.000,C 90.000,E1 126.503} C_DIS
LIN {X 0.081,Y -312.365,Z 980.700,A 0.000,B 0.000,C 90.000,E1 125.964} C_DIS
LIN {X 0.049,Y -313.975,Z 980.698,A 0.000,B 0.000,C 90.000,E1 125.644} C_DIS
LIN {X 0.090,Y -315.239,Z 980.696,A 0.000,B 0.000,C 90.000,E1 125.311} C_DIS
LIN {X -0.048,Y -325.892,Z 980.678,A 0.000,B 0.000,C 90.000,E1 122.133} C_DIS
LIN {X 0.068,Y -336.811,Z 980.663,A 0.000,B 0.000,C 90.000,E1 119.283} C_DIS
LIN {X 0.178,Y -349.122,Z 980.647,A 0.000,B 0.000,C 90.000,E1 116.488} C_DIS
LIN {X -0.149,Y -362.925,Z 980.632,A 0.000,B 0.000,C 90.000,E1 113.823} C_DIS
LIN {X 0.180,Y -376.549,Z 980.619,A 0.000,B 0.000,C 90.000,E1 111.408} C_DIS
LIN {X -0.126,Y -391.549,Z 980.606,A 0.000,B 0.000,C 90.000,E1 109.141} C_DIS
LIN {X 0.050,Y -408.031,Z 980.594,A 0.000,B 0.000,C 90.000,E1 106.858} C_DIS
LIN {X 0.025,Y -426.113,Z 980.581,A 0.000,B 0.000,C 90.000,E1 104.662} C_DIS
LIN {X 0.068,Y -445.733,Z 980.570,A 0.000,B 0.000,C 90.000,E1 102.535} C_DIS
LIN {X -0.132,Y -466.058,Z 980.559,A 0.000,B 0.000,C 90.000,E1 100.602} C_DIS
LIN {X -0.121,Y -468.406,Z 980.557,A 0.000,B 0.000,C 90.000,E1 100.366} C_DIS
LIN {X 0.159,Y -470.263,Z 980.556,A 0.000,B 0.000,C 90.000,E1 100.084} C_DIS
LIN {X 0.061,Y -471.666,Z 980.555,A 0.000,B 0.000,C 90.000,E1 99.849} C_DIS
LIN {X 0.239,Y -473.507,Z 980.552,A 0.000,B 0.000,C 90.000,E1 99.321} C_DIS
LIN {X -0.122,Y -474.250,Z 980.549,A 0.000,B 0.000,C 90.000,E1 98.859} C_DIS
LIN {X 0.000,Y -474.026,Z 980.546,A 0.000,B 0.000,C 90.000,E1 98.341} C_DIS
LIN {X 0.192,Y -472.802,Z 980.544,A 0.000,B 0.000,C 90.000,E1 97.814} C_DIS
LIN {X -0.012,Y -471.759,Z 980.542,A 0.000,B 0.000,C 90.000,E1 97.587} C_DIS
LIN {X -0.152,Y -470.359,Z 980.541,A 0.000,B 0.000,C 90.000,E1 97.352} C_DIS
LIN {X 0.178,Y -456.773,Z 980.529,A 0.000,B 0.000,C 90.000,E1 95.277} C_DIS
LIN {X -0.079,Y -444.702,Z 980.519,A 0.000,B 0.000,C 90.000,E1 93.498} C_DIS
LIN {X -0.109,Y -428.064,Z 980.505,A 0.000,B 0.000,C 90.000,E1 90.859} C_DIS
LIN {X -0.097,Y -411.480,Z 980.488,A 0.000,B 0.000,C 90.000,E1 87.879} C_DIS
LIN {X -0.052,Y -402.518,Z 980.479,A 0.000,B 0.000,C 90.000,E1 86.216} C_DIS
LIN {X -0.091,Y -391.835,Z 980.468,A 0.000,B 0.000,C 90.000,E1 84.261} C_DIS
LIN {X 0.075,Y -380.845,Z 980.457,A 0.000,B 0.000,C 90.000,E1 82.243} C_DIS
LIN {X 0.111,Y -371.253,Z 980.447,A 0.000,B 0.000,C 90.000,E1 80.500} C_DIS
LIN {X -0.026,Y -361.275,Z 980.438,A 0.000,B 0.000,C 90.000,E1 78.757} C_DIS
LIN {X 0.088,Y -349.541,Z 980.426,A 0.000,B 0.000,C 90.000,E1 76.645} C_DIS
LIN {X 0.107,Y -331.825,Z 980.407,A 0.000,B 0.000,C 90.000,E1 73.268} C_DIS
LIN {X -0.089,Y -319.484,Z 980.393,A 0.000,B 0.000,C 90.000,E1 70.786} C_DIS
LIN {X -0.085,Y -308.938,Z 980.381,A 0.000,B 0.000,C 90.000,E1 68.539} C_DIS
LIN {X -0.088,Y -297.038,Z 980.366,A 0.000,B 0.000,C 90.000,E1 65.921} C_DIS
LIN {X -0.134,Y -285.333,Z 980.351,A 0.000,B 0.000,C 90.000,E1 63.256} C_DIS
LIN {X -0.023,Y -275.157,Z 980.338,A 0.000,B 0.000,C 90.000,E1 60.845} C_DIS
LIN {X -0.089,Y -263.807,Z 980.323,A 0.000,B 0.000,C 90.000,E1 58.074} C_DIS
LIN {X -0.011,Y -251.469,Z 980.305,A 0.000,B 0.000,C 90.000,E1 54.848} C_DIS
LIN {X 0.102,Y -239.807,Z 980.286,A 0.000,B 0.000,C 90.000,E1 51.537} C_DIS
LIN {X 0.044,Y -230.134,Z 980.270,A 0.000,B 0.000,C 90.000,E1 48.566} C_DIS
LIN {X -0.052,Y -219.894,Z 980.251,A 0.000,B 0.000,C 90.000,E1 45.162} C_DIS
LIN {X -0.085,Y -210.368,Z 980.231,A 0.000,B 0.000,C 90.000,E1 41.676} C_DIS
LIN {X 0.090,Y -202.472,Z 980.214,A 0.000,B 0.000,C 90.000,E1 38.463} C_DIS
LIN {X 0.017,Y -195.294,Z 980.196,A 0.000,B 0.000,C 90.000,E1 35.264} C_DIS
LIN {X -0.019,Y -188.783,Z 980.178,A 0.000,B 0.000,C 90.000,E1 32.005} C_DIS
LIN {X -0.033,Y -183.005,Z 980.159,A 0.000,B 0.000,C 90.000,E1 28.693} C_DIS
LIN {X -0.042,Y -177.946,Z 980.141,A 0.000,B 0.000,C 90.000,E1 25.335} C_DIS
LIN {X 0.077,Y -173.686,Z 980.122,A 0.000,B 0.000,C 90.000,E1 21.897} C_DIS
LIN {X 0.002,Y -170.051,Z 980.103,A 0.000,B 0.000,C 90.000,E1 18.489} C_DIS
LIN {X -0.045,Y -166.557,Z 980.079,A 0.000,B 0.000,C 90.000,E1 14.175} C_DIS
LIN {X 0.010,Y -163.736,Z 980.050,A 0.000,B 0.000,C 90.000,E1 8.916} C_DIS
LIN {X 0.035,Y -164.519,Z 979.953,A 0.000,B 0.000,C 90.000,E1 351.602} C_DIS
LIN {X 0.034,Y -167.248,Z 979.929,A 0.000,B 0.000,C 90.000,E1 347.229} C_DIS
LIN {X 0.066,Y -170.236,Z 979.910,A 0.000,B 0.000,C 90.000,E1 343.740} C_DIS
LIN {X -0.019,Y -174.019,Z 979.891,A 0.000,B 0.000,C 90.000,E1 340.315} C_DIS
LIN {X 0.057,Y -178.573,Z 979.872,A 0.000,B 0.000,C 90.000,E1 336.869} C_DIS
LIN {X -0.030,Y -183.853,Z 979.853,A 0.000,B 0.000,C 90.000,E1 333.512} C_DIS
LIN {X 0.106,Y -189.892,Z 979.834,A 0.000,B 0.000,C 90.000,E1 330.127} C_DIS
LIN {X 0.093,Y -196.595,Z 979.816,A 0.000,B 0.000,C 90.000,E1 326.834} C_DIS
LIN {X -0.034,Y -203.789,Z 979.798,A 0.000,B 0.000,C 90.000,E1 323.623} C_DIS
LIN {X -0.073,Y -211.556,Z 979.780,A 0.000,B 0.000,C 90.000,E1 320.436} C_DIS
LIN {X -0.119,Y -219.776,Z 979.763,A 0.000,B 0.000,C 90.000,E1 317.310} C_DIS
LIN {X 0.033,Y -228.754,Z 979.746,A 0.000,B 0.000,C 90.000,E1 314.190} C_DIS
LIN {X 0.071,Y -235.140,Z 979.735,A 0.000,B 0.000,C 90.000,E1 312.285} C_DIS
LIN {X -0.115,Y -242.381,Z 979.725,A 0.000,B 0.000,C 90.000,E1 310.458} C_DIS
LIN {X 0.004,Y -252.096,Z 979.712,A 0.000,B 0.000,C 90.000,E1 308.222} C_DIS
LIN {X -0.107,Y -264.832,Z 979.698,A 0.000,B 0.000,C 90.000,E1 305.724} C_DIS
LIN {X 0.078,Y -280.918,Z 979.683,A 0.000,B 0.000,C 90.000,E1 302.880} C_DIS
LIN {X -0.160,Y -298.305,Z 979.668,A 0.000,B 0.000,C 90.000,E1 300.207} C_DIS
LIN {X 0.110,Y -314.673,Z 979.655,A 0.000,B 0.000,C 90.000,E1 297.847} C_DIS
LIN {X -0.002,Y -327.371,Z 979.646,A 0.000,B 0.000,C 90.000,E1 296.283} C_DIS
LIN {X -0.091,Y -351.520,Z 979.631,A 0.000,B 0.000,C 90.000,E1 293.643} C_DIS
LIN {X 0.181,Y -370.355,Z 979.621,A 0.000,B 0.000,C 90.000,E1 291.716} C_DIS
LIN {X 0.045,Y -389.207,Z 979.611,A 0.000,B 0.000,C 90.000,E1 289.939} C_DIS
LIN {X -0.005,Y -402.442,Z 979.604,A 0.000,B 0.000,C 90.000,E1 288.671} C_DIS
LIN {X -0.048,Y -412.749,Z 979.598,A 0.000,B 0.000,C 90.000,E1 287.638} C_DIS
LIN {X 0.049,Y -422.669,Z 979.592,A 0.000,B 0.000,C 90.000,E1 286.567} C_DIS
LIN {X 0.109,Y -432.365,Z 979.586,A 0.000,B 0.000,C 90.000,E1 285.481} C_DIS
LIN {X -0.189,Y -439.232,Z 979.582,A 0.000,B 0.000,C 90.000,E1 284.717} C_DIS
LIN {X -0.096,Y -447.926,Z 979.576,A 0.000,B 0.000,C 90.000,E1 283.647} C_DIS
LIN {X -0.004,Y -456.071,Z 979.570,A 0.000,B 0.000,C 90.000,E1 282.591} C_DIS
LIN {X 0.189,Y -463.624,Z 979.564,A 0.000,B 0.000,C 90.000,E1 281.535} C_DIS
LIN {X -0.079,Y -470.579,Z 979.559,A 0.000,B 0.000,C 90.000,E1 280.546} C_DIS
LIN {X -0.128,Y -475.299,Z 979.554,A 0.000,B 0.000,C 90.000,E1 279.792} C_DIS
LIN {X -0.064,Y -479.408,Z 979.550,A 0.000,B 0.000,C 90.000,E1 279.029} C_DIS
LIN {X -0.039,Y -482.890,Z 979.546,A 0.000,B 0.000,C 90.000,E1 278.276} C_DIS
LIN {X -0.050,Y -485.761,Z 979.542,A 0.000,B 0.000,C 90.000,E1 277.530} C_DIS
LIN {X 0.139,Y -487.325,Z 979.539,A 0.000,B 0.000,C 90.000,E1 277.011} C_DIS
LIN {X -0.090,Y -488.583,Z 979.536,A 0.000,B 0.000,C 90.000,E1 276.543} C_DIS
LIN {X 0.064,Y -489.468,Z 979.534,A 0.000,B 0.000,C 90.000,E1 276.030} C_DIS
LIN {X -0.207,Y -490.062,Z 979.531,A 0.000,B 0.000,C 90.000,E1 275.568} C_DIS
LIN {X 0.013,Y -490.314,Z 979.528,A 0.000,B 0.000,C 90.000,E1 275.049} C_DIS
LIN {X 0.235,Y -490.192,Z 979.525,A 0.000,B 0.000,C 90.000,E1 274.531} C_DIS
LIN {X -0.067,Y -489.598,Z 979.523,A 0.000,B 0.000,C 90.000,E1 274.073} C_DIS
LIN {X 0.154,Y -488.474,Z 979.520,A 0.000,B 0.000,C 90.000,E1 273.555} C_DIS
LIN {X -0.120,Y -486.837,Z 979.517,A 0.000,B 0.000,C 90.000,E1 273.094} C_DIS
LIN {X 0.059,Y -484.495,Z 979.514,A 0.000,B 0.000,C 90.000,E1 272.579} C_DIS
LIN {X 0.225,Y -481.483,Z 979.512,A 0.000,B 0.000,C 90.000,E1 272.064} C_DIS
LIN {X -0.089,Y -477.599,Z 979.509,A 0.000,B 0.000,C 90.000,E1 271.604} C_DIS
LIN {X 0.042,Y -472.708,Z 979.506,A 0.000,B 0.000,C 90.000,E1 271.088} C_DIS
LIN {X -0.166,Y -466.898,Z 979.503,A 0.000,B 0.000,C 90.000,E1 270.630} C_DIS
LIN {X 0.100,Y -460.724,Z 979.501,A 0.000,B 0.000,C 90.000,E1 270.172} C_DIS
LIN {X -0.133,Y -454.110,Z 979.499,A 0.000,B 0.000,C 90.000,E1 269.828} C_DIS
LIN {X 0.080,Y -447.218,Z 979.497,A 0.000,B 0.000,C 90.000,E1 269.484} C_DIS
LIN {X -0.184,Y -439.882,Z 979.496,A 0.000,B 0.000,C 90.000,E1 269.255} C_DIS
LIN {X -0.037,Y -432.308,Z 979.495,A 0.000,B 0.000,C 90.000,E1 269.026} C_DIS
LIN {X 0.010,Y -424.406,Z 979.494,A 0.000,B 0.000,C 90.000,E1 268.854} C_DIS
LIN {X -0.078,Y -415.817,Z 979.493,A 0.000,B 0.000,C 90.000,E1 268.740} C_DIS
LIN {X -0.176,Y -408.071,Z 979.493,A 0.000,B 0.000,C 90.000,E1 268.682} C_DIS
LIN {X 0.010,Y -399.948,Z 979.492,A 0.000,B 0.000,C 90.000,E1 268.625} C_DIS
LIN {X -0.019,Y -181.238,Z 979.492,A 0.000,B 0.000,C 90.000,E1 268.625} C_DIS
LIN {X 0.080,Y -180.896,Z 979.473,A 0.000,B 0.000,C 90.000,E1 265.179} C_DIS
LIN {X -0.092,Y -179.842,Z 979.459,A 0.000,B 0.000,C 90.000,E1 262.704} C_DIS
LIN {X -0.036,Y -179.026,Z 979.445,A 0.000,B 0.000,C 90.000,E1 260.151} C_DIS
LIN {X 0.027,Y -178.671,Z 979.441,A 0.000,B 0.000,C 90.000,E1 259.285} C_DIS
LIN {X -0.038,Y -175.721,Z 979.412,A 0.000,B 0.000,C 90.000,E1 254.212} C_DIS
LIN {X -0.020,Y -172.438,Z 979.388,A 0.000,B 0.000,C 90.000,E1 249.934} C_DIS
LIN {X -0.066,Y -171.268,Z 979.379,A 0.000,B 0.000,C 90.000,E1 248.230} C_DIS
LIN {X -0.020,Y -167.538,Z 979.355,A 0.000,B 0.000,C 90.000,E1 243.896} C_DIS
LIN {X -0.006,Y -166.153,Z 979.345,A 0.000,B 0.000,C 90.000,E1 242.153} C_DIS
LIN {X -0.015,Y -162.930,Z 979.326,A 0.000,B 0.000,C 90.000,E1 238.663} C_DIS
LIN {X -0.038,Y -161.601,Z 979.316,A 0.000,B 0.000,C 90.000,E1 236.914} C_DIS
LIN {X -0.061,Y -159.125,Z 979.301,A 0.000,B 0.000,C 90.000,E1 234.276} C_DIS
LIN {X -0.050,Y -155.648,Z 979.277,A 0.000,B 0.000,C 90.000,E1 229.828} C_DIS
LIN {X 0.002,Y -151.919,Z 979.252,A 0.000,B 0.000,C 90.000,E1 225.324} C_DIS
LIN {X 0.018,Y -150.154,Z 979.237,A 0.000,B 0.000,C 90.000,E1 222.609} C_DIS
LIN {X -0.062,Y -146.936,Z 979.211,A 0.000,B 0.000,C 90.000,E1 218.096} C_DIS
LIN {X 0.046,Y -145.523,Z 979.196,A 0.000,B 0.000,C 90.000,E1 215.311} C_DIS
LIN {X 0.039,Y -142.923,Z 979.171,A 0.000,B 0.000,C 90.000,E1 210.718} C_DIS
LIN {X -0.034,Y -141.545,Z 979.150,A 0.000,B 0.000,C 90.000,E1 207.052} C_DIS
LIN {X -0.045,Y -139.403,Z 979.114,A 0.000,B 0.000,C 90.000,E1 200.556} C_DIS
LIN {X 0.009,Y -139.121,Z 979.104,A 0.000,B 0.000,C 90.000,E1 198.671} C_DIS
LIN {X 0.040,Y -138.352,Z 979.057,A 0.000,B 0.000,C 90.000,E1 190.254} C_DIS
LIN {X 0.030,Y -139.502,Z 979.005,A 0.000,B 0.000,C 90.000,E1 180.917} C_DIS
LIN {X -0.029,Y -141.133,Z 978.974,A 0.000,B 0.000,C 90.000,E1 175.355} C_DIS
LIN {X -0.076,Y -142.514,Z 978.959,A 0.000,B 0.000,C 90.000,E1 172.591} C_DIS
LIN {X 0.011,Y -144.773,Z 978.933,A 0.000,B 0.000,C 90.000,E1 167.937} C_DIS
LIN {X -0.040,Y -147.388,Z 978.913,A 0.000,B 0.000,C 90.000,E1 164.283} C_DIS
LIN {X 0.023,Y -150.717,Z 978.887,A 0.000,B 0.000,C 90.000,E1 159.699} C_DIS
LIN {X -0.037,Y -154.198,Z 978.867,A 0.000,B 0.000,C 90.000,E1 156.102} C_DIS
LIN {X 0.033,Y -157.638,Z 978.847,A 0.000,B 0.000,C 90.000,E1 152.487} C_DIS
LIN {X -0.020,Y -161.896,Z 978.827,A 0.000,B 0.000,C 90.000,E1 148.948} C_DIS
LIN {X 0.088,Y -166.086,Z 978.808,A 0.000,B 0.000,C 90.000,E1 145.388} C_DIS
LIN {X 0.087,Y -171.095,Z 978.789,A 0.000,B 0.000,C 90.000,E1 141.904} C_DIS
LIN {X 0.006,Y -175.968,Z 978.769,A 0.000,B 0.000,C 90.000,E1 138.485} C_DIS
LIN {X 0.121,Y -180.213,Z 978.755,A 0.000,B 0.000,C 90.000,E1 135.891} C_DIS
LIN {X 0.095,Y -185.629,Z 978.736,A 0.000,B 0.000,C 90.000,E1 132.528} C_DIS
LIN {X -0.119,Y -190.224,Z 978.723,A 0.000,B 0.000,C 90.000,E1 130.092} C_DIS
LIN {X 0.005,Y -195.400,Z 978.706,A 0.000,B 0.000,C 90.000,E1 127.076} C_DIS
LIN {X -0.045,Y -299.109,Z 978.706,A 0.000,B 0.000,C 90.000,E1 127.076} C_DIS
LIN {X 0.088,Y -300.442,Z 978.706,A 0.000,B 0.000,C 90.000,E1 127.030} C_DIS
LIN {X 0.085,Y -306.194,Z 978.704,A 0.000,B 0.000,C 90.000,E1 126.744} C_DIS
LIN {X -0.036,Y -309.284,Z 978.703,A 0.000,B 0.000,C 90.000,E1 126.457} C_DIS
LIN {X 0.015,Y -312.911,Z 978.699,A 0.000,B 0.000,C 90.000,E1 125.884} C_DIS
LIN {X -0.199,Y -314.374,Z 978.698,A 0.000,B 0.000,C 90.000,E1 125.598} C_DIS
LIN {X -0.051,Y -318.567,Z 978.690,A 0.000,B 0.000,C 90.000,E1 124.278} C_DIS
LIN {X 0.020,Y -329.703,Z 978.673,A 0.000,B 0.000,C 90.000,E1 121.082} C_DIS
LIN {X -0.047,Y -341.121,Z 978.657,A 0.000,B 0.000,C 90.000,E1 118.281} C_DIS
LIN {X -0.136,Y -353.960,Z 978.642,A 0.000,B 0.000,C 90.000,E1 115.540} C_DIS
LIN {X -0.082,Y -366.663,Z 978.628,A 0.000,B 0.000,C 90.000,E1 113.131} C_DIS
LIN {X -0.149,Y -380.670,Z 978.615,A 0.000,B 0.000,C 90.000,E1 110.791} C_DIS
LIN {X -0.123,Y -396.082,Z 978.603,A 0.000,B 0.000,C 90.000,E1 108.489} C_DIS
LIN {X 0.180,Y -413.009,Z 978.590,A 0.000,B 0.000,C 90.000,E1 106.205} C_DIS
LIN {X -0.132,Y -431.571,Z 978.578,A 0.000,B 0.000,C 90.000,E1 104.064} C_DIS
LIN {X 0.124,Y -451.462,Z 978.566,A 0.000,B 0.000,C 90.000,E1 101.951} C_DIS
LIN {X -0.224,Y -466.771,Z 978.558,A 0.000,B 0.000,C 90.000,E1 100.546} C_DIS
LIN {X -0.208,Y -468.939,Z 978.557,A 0.000,B 0.000,C 90.000,E1 100.310} C_DIS
LIN {X 0.102,Y -470.704,Z 978.556,A 0.000,B 0.000,C 90.000,E1 100.018} C_DIS
LIN {X -0.133,Y -472.029,Z 978.554,A 0.000,B 0.000,C 90.000,E1 99.792} C_DIS
LIN {X 0.046,Y -473.685,Z 978.552,A 0.000,B 0.000,C 90.000,E1 99.265} C_DIS
LIN {X 0.158,Y -474.277,Z 978.549,A 0.000,B 0.000,C 90.000,E1 98.746} C_DIS
LIN {X -0.120,Y -473.906,Z 978.546,A 0.000,B 0.000,C 90.000,E1 98.276} C_DIS
LIN {X 0.005,Y -472.517,Z 978.543,A 0.000,B 0.000,C 90.000,E1 97.757} C_DIS
LIN {X -0.198,Y -471.372,Z 978.542,A 0.000,B 0.000,C 90.000,E1 97.530} C_DIS
LIN {X -0.022,Y -468.131,Z 978.539,A 0.000,B 0.000,C 90.000,E1 97.004} C_DIS
LIN {X -0.012,Y -456.270,Z 978.529,A 0.000,B 0.000,C 90.000,E1 95.220} C_DIS
LIN {X 0.171,Y -444.232,Z 978.519,A 0.000,B 0.000,C 90.000,E1 93.383} C_DIS
LIN {X 0.120,Y -427.642,Z 978.504,A 0.000,B 0.000,C 90.000,E1 90.745} C_DIS
LIN {X 0.111,Y -411.067,Z 978.488,A 0.000,B 0.000,C 90.000,E1 87.764} C_DIS
LIN {X 0.142,Y -402.066,Z 978.478,A 0.000,B 0.000,C 90.000,E1 86.102} C_DIS
LIN {X 0.085,Y -391.376,Z 978.468,A 0.000,B 0.000,C 90.000,E1 84.147} C_DIS
LIN {X -0.143,Y -380.391,Z 978.456,A 0.000,B 0.000,C 90.000,E1 82.186} C_DIS
LIN {X -0.111,Y -370.756,Z 978.447,A 0.000,B 0.000,C 90.000,E1 80.443} C_DIS
LIN {X 0.173,Y -360.789,Z 978.437,A 0.000,B 0.000,C 90.000,E1 78.634} C_DIS
LIN {X -0.125,Y -347.364,Z 978.424,A 0.000,B 0.000,C 90.000,E1 76.284} C_DIS
LIN {X -0.039,Y -331.334,Z 978.407,A 0.000,B 0.000,C 90.000,E1 73.196} C_DIS
LIN {X -0.036,Y -319.039,Z 978.393,A 0.000,B 0.000,C 90.000,E1 70.678} C_DIS
LIN {X 0.061,Y -308.486,Z 978.380,A 0.000,B 0.000,C 90.000,E1 68.411} C_DIS
LIN {X 0.045,Y -296.600,Z 978.366,A 0.000,B 0.000,C 90.000,E1 65.793} C_DIS
LIN {X 0.009,Y -286.355,Z 978.353,A 0.000,B 0.000,C 90.000,E1 63.461} C_DIS
LIN {X 0.128,Y -276.140,Z 978.339,A 0.000,B 0.000,C 90.000,E1 61.051} C_DIS
LIN {X 0.076,Y -264.749,Z 978.324,A 0.000,B 0.000,C 90.000,E1 58.280} C_DIS
LIN {X -0.030,Y -252.368,Z 978.306,A 0.000,B 0.000,C 90.000,E1 55.102} C_DIS
LIN {X -0.034,Y -240.637,Z 978.288,A 0.000,B 0.000,C 90.000,E1 51.823} C_DIS
LIN {X 0.050,Y -229.772,Z 978.269,A 0.000,B 0.000,C 90.000,E1 48.447} C_DIS
LIN {X 0.110,Y -219.575,Z 978.250,A 0.000,B 0.000,C 90.000,E1 45.000} C_DIS
LIN {X 0.061,Y -210.089,Z 978.231,A 0.000,B 0.000,C 90.000,E1 41.515} C_DIS
LIN {X -0.063,Y -202.247,Z 978.213,A 0.000,B 0.000,C 90.000,E1 38.382} C_DIS
LIN {X -0.026,Y -195.102,Z 978.195,A 0.000,B 0.000,C 90.000,E1 35.152} C_DIS
LIN {X -0.017,Y -188.622,Z 978.177,A 0.000,B 0.000,C 90.000,E1 31.878} C_DIS
LIN {X -0.033,Y -182.888,Z 978.159,A 0.000,B 0.000,C 90.000,E1 28.565} C_DIS
LIN {X -0.045,Y -177.860,Z 978.140,A 0.000,B 0.000,C 90.000,E1 25.207} C_DIS
LIN {X 0.071,Y -173.633,Z 978.121,A 0.000,B 0.000,C 90.000,E1 21.770} C_DIS
LIN {X -0.008,Y -170.024,Z 978.102,A 0.000,B 0.000,C 90.000,E1 18.362} C_DIS
LIN {X 0.061,Y -166.560,Z 978.078,A 0.000,B 0.000,C 90.000,E1 14.008} C_DIS
LIN {X -0.038,Y -163.771,Z 978.049,A 0.000,B 0.000,C 90.000,E1 8.803} C_DIS
LIN {X 0.070,Y -164.214,Z 977.958,A 0.000,B 0.000,C 90.000,E1 352.470} C_DIS
LIN {X -0.004,Y -166.749,Z 977.934,A 0.000,B 0.000,C 90.000,E1 348.117} C_DIS
LIN {X 0.012,Y -169.563,Z 977.915,A 0.000,B 0.000,C 90.000,E1 344.629} C_DIS
LIN {X 0.025,Y -173.150,Z 977.895,A 0.000,B 0.000,C 90.000,E1 341.167} C_DIS
LIN {X 0.015,Y -177.514,Z 977.876,A 0.000,B 0.000,C 90.000,E1 337.741} C_DIS
LIN {X 0.065,Y -182.623,Z 977.858,A 0.000,B 0.000,C 90.000,E1 334.332} C_DIS
LIN {X -0.005,Y -188.455,Z 977.839,A 0.000,B 0.000,C 90.000,E1 331.001} C_DIS
LIN {X -0.060,Y -195.030,Z 977.820,A 0.000,B 0.000,C 90.000,E1 327.709} C_DIS
LIN {X 0.104,Y -202.082,Z 977.802,A 0.000,B 0.000,C 90.000,E1 324.402} C_DIS
LIN {X 0.085,Y -210.691,Z 977.782,A 0.000,B 0.000,C 90.000,E1 320.803} C_DIS
LIN {X -0.068,Y -219.911,Z 977.763,A 0.000,B 0.000,C 90.000,E1 317.310} C_DIS
LIN {X 0.091,Y -228.945,Z 977.746,A 0.000,B 0.000,C 90.000,E1 314.190} C_DIS
LIN {X 0.091,Y -236.717,Z 977.733,A 0.000,B 0.000,C 90.000,E1 311.919} C_DIS
LIN {X -0.079,Y -245.651,Z 977.721,A 0.000,B 0.000,C 90.000,E1 309.725} C_DIS
LIN {X -0.063,Y -253.952,Z 977.710,A 0.000,B 0.000,C 90.000,E1 307.890} C_DIS
LIN {X 0.021,Y -266.858,Z 977.696,A 0.000,B 0.000,C 90.000,E1 305.358} C_DIS
LIN {X 0.013,Y -280.971,Z 977.683,A 0.000,B 0.000,C 90.000,E1 302.911} C_DIS
LIN {X -0.068,Y -298.323,Z 977.668,A 0.000,B 0.000,C 90.000,E1 300.207} C_DIS
LIN {X -0.071,Y -314.639,Z 977.655,A 0.000,B 0.000,C 90.000,E1 297.897} C_DIS
LIN {X 0.052,Y -327.378,Z 977.646,A 0.000,B 0.000,C 90.000,E1 296.283} C_DIS
LIN {X 0.140,Y -351.185,Z 977.631,A 0.000,B 0.000,C 90.000,E1 293.643} C_DIS
LIN {X -0.051,Y -370.160,Z 977.621,A 0.000,B 0.000,C 90.000,E1 291.770} C_DIS
LIN {X 0.098,Y -386.541,Z 977.612,A 0.000,B 0.000,C 90.000,E1 290.174} C_DIS
LIN {X 0.001,Y -399.910,Z 977.605,A 0.000,B 0.000,C 90.000,E1 288.906} C_DIS
LIN {X -0.050,Y -410.311,Z 977.599,A 0.000,B 0.000,C 90.000,E1 287.873} C_DIS
LIN {X 0.150,Y -420.228,Z 977.593,A 0.000,B 0.000,C 90.000,E1 286.804} C_DIS
LIN {X 0.071,Y -430.027,Z 977.587,A 0.000,B 0.000,C 90.000,E1 285.733} C_DIS
LIN {X 0.065,Y -439.271,Z 977.581,A 0.000,B 0.000,C 90.000,E1 284.662} C_DIS
LIN {X 0.165,Y -447.905,Z 977.576,A 0.000,B 0.000,C 90.000,E1 283.592} C_DIS
LIN {X -0.181,Y -456.031,Z 977.570,A 0.000,B 0.000,C 90.000,E1 282.591} C_DIS
LIN {X 0.007,Y -463.628,Z 977.564,A 0.000,B 0.000,C 90.000,E1 281.535} C_DIS
LIN {X 0.201,Y -470.623,Z 977.558,A 0.000,B 0.000,C 90.000,E1 280.489} C_DIS
LIN {X 0.235,Y -475.367,Z 977.554,A 0.000,B 0.000,C 90.000,E1 279.726} C_DIS
LIN {X 0.223,Y -479.502,Z 977.550,A 0.000,B 0.000,C 90.000,E1 278.973} C_DIS
LIN {X 0.253,Y -483.019,Z 977.546,A 0.000,B 0.000,C 90.000,E1 278.219} C_DIS
LIN {X -0.237,Y -485.872,Z 977.542,A 0.000,B 0.000,C 90.000,E1 277.530} C_DIS
LIN {X 0.011,Y -487.452,Z 977.539,A 0.000,B 0.000,C 90.000,E1 277.004} C_DIS
LIN {X 0.209,Y -488.698,Z 977.536,A 0.000,B 0.000,C 90.000,E1 276.486} C_DIS
LIN {X -0.122,Y -489.606,Z 977.533,A 0.000,B 0.000,C 90.000,E1 276.030} C_DIS
LIN {X 0.094,Y -490.159,Z 977.531,A 0.000,B 0.000,C 90.000,E1 275.511} C_DIS
LIN {X -0.172,Y -490.388,Z 977.528,A 0.000,B 0.000,C 90.000,E1 275.049} C_DIS
LIN {X 0.050,Y -490.265,Z 977.525,A 0.000,B 0.000,C 90.000,E1 274.531} C_DIS
LIN {X -0.216,Y -489.662,Z 977.522,A 0.000,B 0.000,C 90.000,E1 274.069} C_DIS
LIN {X -0.030,Y -488.530,Z 977.520,A 0.000,B 0.000,C 90.000,E1 273.555} C_DIS
LIN {X 0.183,Y -486.856,Z 977.517,A 0.000,B 0.000,C 90.000,E1 273.037} C_DIS
LIN {X -0.122,Y -484.538,Z 977.514,A 0.000,B 0.000,C 90.000,E1 272.579} C_DIS
LIN {X 0.044,Y -481.463,Z 977.511,A 0.000,B 0.000,C 90.000,E1 272.064} C_DIS
LIN {X -0.119,Y -479.668,Z 977.510,A 0.000,B 0.000,C 90.000,E1 271.835} C_DIS
LIN {X 0.036,Y -475.209,Z 977.507,A 0.000,B 0.000,C 90.000,E1 271.318} C_DIS
LIN {X -0.135,Y -472.665,Z 977.506,A 0.000,B 0.000,C 90.000,E1 271.088} C_DIS
LIN {X 0.094,Y -466.770,Z 977.503,A 0.000,B 0.000,C 90.000,E1 270.573} C_DIS
LIN {X -0.108,Y -460.517,Z 977.501,A 0.000,B 0.000,C 90.000,E1 270.172} C_DIS
LIN {X 0.169,Y -453.975,Z 977.499,A 0.000,B 0.000,C 90.000,E1 269.771} C_DIS
LIN {X -0.039,Y -447.116,Z 977.497,A 0.000,B 0.000,C 90.000,E1 269.484} C_DIS
LIN {X 0.155,Y -439.951,Z 977.496,A 0.000,B 0.000,C 90.000,E1 269.198} C_DIS
LIN {X -0.167,Y -432.181,Z 977.494,A 0.000,B 0.000,C 90.000,E1 269.026} C_DIS
LIN {X -0.114,Y -424.294,Z 977.494,A 0.000,B 0.000,C 90.000,E1 268.854} C_DIS
LIN {X -0.199,Y -416.006,Z 977.493,A 0.000,B 0.000,C 90.000,E1 268.740} C_DIS
LIN {X 0.103,Y -408.216,Z 977.492,A 0.000,B 0.000,C 90.000,E1 268.625} C_DIS
LIN {X -0.118,Y -397.302,Z 977.492,A 0.000,B 0.000,C 90.000,E1 268.625} C_DIS
LIN {X -0.077,Y -181.234,Z 977.492,A 0.000,B 0.000,C 90.000,E1 268.625} C_DIS
LIN {X 0.027,Y -180.895,Z 977.473,A 0.000,B 0.000,C 90.000,E1 265.179} C_DIS
LIN {X -0.073,Y -179.520,Z 977.455,A 0.000,B 0.000,C 90.000,E1 261.837} C_DIS
LIN {X 0.089,Y -179.022,Z 977.445,A 0.000,B 0.000,C 90.000,E1 260.095} C_DIS
LIN {X -0.025,Y -178.661,Z 977.440,A 0.000,B 0.000,C 90.000,E1 259.285} C_DIS
LIN {X 0.081,Y -175.711,Z 977.412,A 0.000,B 0.000,C 90.000,E1 254.157} C_DIS
LIN {X -0.071,Y -172.426,Z 977.388,A 0.000,B 0.000,C 90.000,E1 249.934} C_DIS
LIN {X 0.107,Y -171.251,Z 977.379,A 0.000,B 0.000,C 90.000,E1 248.156} C_DIS
LIN {X -0.069,Y -167.525,Z 977.355,A 0.000,B 0.000,C 90.000,E1 243.896} C_DIS
LIN {X 0.015,Y -166.920,Z 977.350,A 0.000,B 0.000,C 90.000,E1 242.999} C_DIS
LIN {X -0.064,Y -162.916,Z 977.326,A 0.000,B 0.000,C 90.000,E1 238.663} C_DIS
LIN {X -0.086,Y -161.590,Z 977.316,A 0.000,B 0.000,C 90.000,E1 236.914} C_DIS
LIN {X 0.041,Y -158.331,Z 977.296,A 0.000,B 0.000,C 90.000,E1 233.336} C_DIS
LIN {X 0.021,Y -155.633,Z 977.277,A 0.000,B 0.000,C 90.000,E1 229.784} C_DIS
LIN {X -0.045,Y -151.907,Z 977.252,A 0.000,B 0.000,C 90.000,E1 225.324} C_DIS
LIN {X -0.028,Y -150.139,Z 977.237,A 0.000,B 0.000,C 90.000,E1 222.609} C_DIS
LIN {X 0.009,Y -146.925,Z 977.211,A 0.000,B 0.000,C 90.000,E1 218.051} C_DIS
LIN {X 0.000,Y -145.513,Z 977.196,A 0.000,B 0.000,C 90.000,E1 215.311} C_DIS
LIN {X -0.006,Y -142.914,Z 977.171,A 0.000,B 0.000,C 90.000,E1 210.718} C_DIS
LIN {X 0.047,Y -141.537,Z 977.150,A 0.000,B 0.000,C 90.000,E1 207.001} C_DIS
LIN {X -0.041,Y -139.400,Z 977.114,A 0.000,B 0.000,C 90.000,E1 200.536} C_DIS
LIN {X -0.035,Y -139.116,Z 977.104,A 0.000,B 0.000,C 90.000,E1 198.671} C_DIS
LIN {X -0.003,Y -138.352,Z 977.057,A 0.000,B 0.000,C 90.000,E1 190.254} C_DIS
LIN {X -0.014,Y -139.506,Z 977.005,A 0.000,B 0.000,C 90.000,E1 180.917} C_DIS
LIN {X -0.073,Y -141.140,Z 976.974,A 0.000,B 0.000,C 90.000,E1 175.355} C_DIS
LIN {X 0.020,Y -142.522,Z 976.959,A 0.000,B 0.000,C 90.000,E1 172.534} C_DIS
LIN {X -0.034,Y -144.785,Z 976.933,A 0.000,B 0.000,C 90.000,E1 167.937} C_DIS
LIN {X -0.046,Y -147.401,Z 976.912,A 0.000,B 0.000,C 90.000,E1 164.267} C_DIS
LIN {X -0.015,Y -149.975,Z 976.892,A 0.000,B 0.000,C 90.000,E1 160.604} C_DIS
LIN {X -0.006,Y -153.299,Z 976.872,A 0.000,B 0.000,C 90.000,E1 156.975} C_DIS
LIN {X -0.018,Y -155.002,Z 976.862,A 0.000,B 0.000,C 90.000,E1 155.177} C_DIS
LIN {X -0.005,Y -158.643,Z 976.842,A 0.000,B 0.000,C 90.000,E1 151.591} C_DIS
LIN {X 0.014,Y -161.918,Z 976.827,A 0.000,B 0.000,C 90.000,E1 148.918} C_DIS
LIN {X 0.039,Y -166.109,Z 976.808,A 0.000,B 0.000,C 90.000,E1 145.388} C_DIS
LIN {X 0.036,Y -171.119,Z 976.788,A 0.000,B 0.000,C 90.000,E1 141.904} C_DIS
LIN {X -0.045,Y -175.995,Z 976.769,A 0.000,B 0.000,C 90.000,E1 138.485} C_DIS
LIN {X 0.068,Y -180.243,Z 976.755,A 0.000,B 0.000,C 90.000,E1 135.891} C_DIS
LIN {X 0.042,Y -185.657,Z 976.736,A 0.000,B 0.000,C 90.000,E1 132.528} C_DIS
LIN {X 0.095,Y -190.256,Z 976.722,A 0.000,B 0.000,C 90.000,E1 130.011} C_DIS
LIN {X 0.107,Y -195.344,Z 976.706,A 0.000,B 0.000,C 90.000,E1 127.076} C_DIS
LIN {X 0.134,Y -299.108,Z 976.706,A 0.000,B 0.000,C 90.000,E1 127.076} C_DIS
LIN {X -0.017,Y -300.722,Z 976.706,A 0.000,B 0.000,C 90.000,E1 127.076} C_DIS
LIN {X -0.040,Y -304.477,Z 976.705,A 0.000,B 0.000,C 90.000,E1 126.916} C_DIS
LIN {X -0.001,Y -306.670,Z 976.704,A 0.000,B 0.000,C 90.000,E1 126.744} C_DIS
LIN {X 0.005,Y -310.560,Z 976.702,A 0.000,B 0.000,C 90.000,E1 126.297} C_DIS
LIN {X -0.134,Y -312.446,Z 976.700,A 0.000,B 0.000,C 90.000,E1 126.011} C_DIS
LIN {X -0.020,Y -313.927,Z 976.698,A 0.000,B 0.000,C 90.000,E1 125.678} C_DIS
LIN {X 0.010,Y -316.150,Z 976.695,A 0.000,B 0.000,C 90.000,E1 125.025} C_DIS
LIN {X 0.167,Y -326.921,Z 976.677,A 0.000,B 0.000,C 90.000,E1 121.799} C_DIS
LIN {X 0.025,Y -337.980,Z 976.661,A 0.000,B 0.000,C 90.000,E1 118.999} C_DIS
LIN {X 0.000,Y -350.440,Z 976.646,A 0.000,B 0.000,C 90.000,E1 116.232} C_DIS
LIN {X 0.034,Y -364.404,Z 976.631,A 0.000,B 0.000,C 90.000,E1 113.515} C_DIS
LIN {X 0.059,Y -378.184,Z 976.618,A 0.000,B 0.000,C 90.000,E1 111.153} C_DIS
LIN {X 0.025,Y -393.351,Z 976.605,A 0.000,B 0.000,C 90.000,E1 108.852} C_DIS
LIN {X -0.129,Y -410.014,Z 976.592,A 0.000,B 0.000,C 90.000,E1 106.622} C_DIS
LIN {X -0.004,Y -428.291,Z 976.580,A 0.000,B 0.000,C 90.000,E1 104.411} C_DIS
LIN {X 0.049,Y -448.034,Z 976.568,A 0.000,B 0.000,C 90.000,E1 102.299} C_DIS
LIN {X 0.002,Y -468.226,Z 976.558,A 0.000,B 0.000,C 90.000,E1 100.366} C_DIS
LIN {X -0.052,Y -470.024,Z 976.556,A 0.000,B 0.000,C 90.000,E1 100.141} C_DIS
LIN {X -0.201,Y -471.516,Z 976.555,A 0.000,B 0.000,C 90.000,E1 99.905} C_DIS
LIN {X 0.114,Y -472.631,Z 976.553,A 0.000,B 0.000,C 90.000,E1 99.613} C_DIS
LIN {X -0.247,Y -473.957,Z 976.551,A 0.000,B 0.000,C 90.000,E1 99.151} C_DIS
LIN {X -0.060,Y -474.268,Z 976.548,A 0.000,B 0.000,C 90.000,E1 98.624} C_DIS
LIN {X 0.063,Y -473.615,Z 976.545,A 0.000,B 0.000,C 90.000,E1 98.106} C_DIS
LIN {X 0.190,Y -471.897,Z 976.542,A 0.000,B 0.000,C 90.000,E1 97.587} C_DIS
LIN {X 0.047,Y -470.543,Z 976.541,A 0.000,B 0.000,C 90.000,E1 97.352} C_DIS
LIN {X -0.078,Y -457.020,Z 976.530,A 0.000,B 0.000,C 90.000,E1 95.334} C_DIS
LIN {X 0.125,Y -445.014,Z 976.520,A 0.000,B 0.000,C 90.000,E1 93.498} C_DIS
LIN {X -0.193,Y -426.794,Z 976.503,A 0.000,B 0.000,C 90.000,E1 90.630} C_DIS
LIN {X 0.105,Y -411.717,Z 976.488,A 0.000,B 0.000,C 90.000,E1 87.879} C_DIS
LIN {X 0.150,Y -402.723,Z 976.479,A 0.000,B 0.000,C 90.000,E1 86.216} C_DIS
LIN {X 0.114,Y -392.025,Z 976.468,A 0.000,B 0.000,C 90.000,E1 84.261} C_DIS
LIN {X -0.133,Y -382.673,Z 976.459,A 0.000,B 0.000,C 90.000,E1 82.591} C_DIS
LIN {X -0.061,Y -373.104,Z 976.449,A 0.000,B 0.000,C 90.000,E1 80.849} C_DIS
LIN {X -0.158,Y -363.218,Z 976.439,A 0.000,B 0.000,C 90.000,E1 79.106} C_DIS
LIN {X 0.003,Y -351.402,Z 976.428,A 0.000,B 0.000,C 90.000,E1 76.992} C_DIS
LIN {X 0.099,Y -333.554,Z 976.409,A 0.000,B 0.000,C 90.000,E1 73.614} C_DIS
LIN {X 0.154,Y -321.228,Z 976.395,A 0.000,B 0.000,C 90.000,E1 71.094} C_DIS
LIN {X 0.106,Y -309.132,Z 976.381,A 0.000,B 0.000,C 90.000,E1 68.539} C_DIS
LIN {X -0.059,Y -298.714,Z 976.368,A 0.000,B 0.000,C 90.000,E1 66.282} C_DIS
LIN {X -0.038,Y -288.429,Z 976.355,A 0.000,B 0.000,C 90.000,E1 63.948} C_DIS
LIN {X 0.006,Y -278.210,Z 976.342,A 0.000,B 0.000,C 90.000,E1 61.563} C_DIS
LIN {X -0.057,Y -265.314,Z 976.325,A 0.000,B 0.000,C 90.000,E1 58.456} C_DIS
LIN {X 0.046,Y -254.237,Z 976.309,A 0.000,B 0.000,C 90.000,E1 55.595} C_DIS
LIN {X -0.059,Y -242.404,Z 976.291,A 0.000,B 0.000,C 90.000,E1 52.351} C_DIS
LIN {X -0.081,Y -231.417,Z 976.272,A 0.000,B 0.000,C 90.000,E1 49.013} C_DIS
LIN {X 0.026,Y -221.159,Z 976.253,A 0.000,B 0.000,C 90.000,E1 45.567} C_DIS
LIN {X 0.025,Y -211.594,Z 976.234,A 0.000,B 0.000,C 90.000,E1 42.081} C_DIS
LIN {X 0.075,Y -203.654,Z 976.216,A 0.000,B 0.000,C 90.000,E1 38.910} C_DIS
LIN {X -0.011,Y -196.409,Z 976.198,A 0.000,B 0.000,C 90.000,E1 35.724} C_DIS
LIN {X -0.026,Y -189.803,Z 976.180,A 0.000,B 0.000,C 90.000,E1 32.467} C_DIS
LIN {X -0.018,Y -183.939,Z 976.162,A 0.000,B 0.000,C 90.000,E1 29.155} C_DIS
LIN {X -0.002,Y -178.794,Z 976.143,A 0.000,B 0.000,C 90.000,E1 25.796} C_DIS
LIN {X 0.051,Y -174.428,Z 976.124,A 0.000,B 0.000,C 90.000,E1 22.386} C_DIS
LIN {X 0.048,Y -170.723,Z 976.105,A 0.000,B 0.000,C 90.000,E1 18.960} C_DIS
LIN {X -0.027,Y -167.089,Z 976.081,A 0.000,B 0.000,C 90.000,E1 14.662} C_DIS
LIN {X -0.044,Y -164.121,Z 976.052,A 0.000,B 0.000,C 90.000,E1 9.434} C_DIS
LIN {X 0.005,Y -162.392,Z 976.004,A 0.000,B 0.000,C 90.000,E1 0.630} C_DIS
LIN {X -0.057,Y -163.958,Z 975.963,A 0.000,B 0.000,C 90.000,E1 353.394} C_DIS
LIN {X 0.006,Y -166.896,Z 975.934,A 0.000,B 0.000,C 90.000,E1 348.117} C_DIS
LIN {X 0.025,Y -169.712,Z 975.915,A 0.000,B 0.000,C 90.000,E1 344.629} C_DIS
LIN {X 0.042,Y -173.303,Z 975.895,A 0.000,B 0.000,C 90.000,E1 341.167} C_DIS
LIN {X 0.036,Y -177.668,Z 975.876,A 0.000,B 0.000,C 90.000,E1 337.741} C_DIS
LIN {X 0.012,Y -182.786,Z 975.858,A 0.000,B 0.000,C 90.000,E1 334.357} C_DIS
LIN {X 0.026,Y -188.624,Z 975.839,A 0.000,B 0.000,C 90.000,E1 331.001} C_DIS
LIN {X -0.024,Y -195.192,Z 975.821,A 0.000,B 0.000,C 90.000,E1 327.709} C_DIS
LIN {X 0.028,Y -202.241,Z 975.802,A 0.000,B 0.000,C 90.000,E1 324.436} C_DIS
LIN {X -0.031,Y -210.832,Z 975.782,A 0.000,B 0.000,C 90.000,E1 320.848} C_DIS
LIN {X -0.014,Y -220.062,Z 975.763,A 0.000,B 0.000,C 90.000,E1 317.310} C_DIS
LIN {X -0.013,Y -229.148,Z 975.746,A 0.000,B 0.000,C 90.000,E1 314.231} C_DIS
LIN {X 0.040,Y -235.548,Z 975.735,A 0.000,B 0.000,C 90.000,E1 312.324} C_DIS
LIN {X 0.008,Y -244.251,Z 975.723,A 0.000,B 0.000,C 90.000,E1 310.092} C_DIS
LIN {X -0.002,Y -252.342,Z 975.713,A 0.000,B 0.000,C 90.000,E1 308.257} C_DIS
LIN {X 0.056,Y -265.027,Z 975.699,A 0.000,B 0.000,C 90.000,E1 305.724} C_DIS
LIN {X -0.133,Y -281.027,Z 975.683,A 0.000,B 0.000,C 90.000,E1 302.959} C_DIS
LIN {X 0.030,Y -298.340,Z 975.668,A 0.000,B 0.000,C 90.000,E1 300.207} C_DIS
LIN {X 0.032,Y -314.602,Z 975.655,A 0.000,B 0.000,C 90.000,E1 297.897} C_DIS
LIN {X 0.016,Y -327.307,Z 975.646,A 0.000,B 0.000,C 90.000,E1 296.309} C_DIS
LIN {X 0.102,Y -353.764,Z 975.630,A 0.000,B 0.000,C 90.000,E1 293.387} C_DIS
LIN {X -0.036,Y -370.103,Z 975.621,A 0.000,B 0.000,C 90.000,E1 291.770} C_DIS
LIN {X 0.126,Y -386.367,Z 975.612,A 0.000,B 0.000,C 90.000,E1 290.174} C_DIS
LIN {X 0.041,Y -399.724,Z 975.605,A 0.000,B 0.000,C 90.000,E1 288.906} C_DIS
LIN {X -0.016,Y -410.123,Z 975.599,A 0.000,B 0.000,C 90.000,E1 287.873} C_DIS
LIN {X 0.038,Y -420.226,Z 975.593,A 0.000,B 0.000,C 90.000,E1 286.804} C_DIS
LIN {X 0.057,Y -430.017,Z 975.587,A 0.000,B 0.000,C 90.000,E1 285.717} C_DIS
LIN {X -0.069,Y -439.253,Z 975.581,A 0.000,B 0.000,C 90.000,E1 284.662} C_DIS
LIN {X 0.029,Y -447.841,Z 975.576,A 0.000,B 0.000,C 90.000,E1 283.592} C_DIS
LIN {X 0.123,Y -455.931,Z 975.570,A 0.000,B 0.000,C 90.000,E1 282.535} C_DIS
LIN {X -0.136,Y -463.581,Z 975.564,A 0.000,B 0.000,C 90.000,E1 281.535} C_DIS
LIN {X 0.053,Y -470.639,Z 975.558,A 0.000,B 0.000,C 90.000,E1 280.489} C_DIS
LIN {X 0.087,Y -475.414,Z 975.554,A 0.000,B 0.000,C 90.000,E1 279.726} C_DIS
LIN {X 0.074,Y -479.569,Z 975.550,A 0.000,B 0.000,C 90.000,E1 278.973} C_DIS
LIN {X 0.103,Y -483.107,Z 975.546,A 0.000,B 0.000,C 90.000,E1 278.219} C_DIS
LIN {X 0.095,Y -485.968,Z 975.542,A 0.000,B 0.000,C 90.000,E1 277.473} C_DIS
LIN {X -0.139,Y -487.536,Z 975.539,A 0.000,B 0.000,C 90.000,E1 277.004} C_DIS
LIN {X 0.059,Y -488.796,Z 975.536,A 0.000,B 0.000,C 90.000,E1 276.486} C_DIS
LIN {X 0.266,Y -489.710,Z 975.533,A 0.000,B 0.000,C 90.000,E1 275.967} C_DIS
LIN {X -0.055,Y -490.265,Z 975.531,A 0.000,B 0.000,C 90.000,E1 275.511} C_DIS
LIN {X 0.168,Y -490.490,Z 975.528,A 0.000,B 0.000,C 90.000,E1 274.992} C_DIS
LIN {X -0.098,Y -490.345,Z 975.525,A 0.000,B 0.000,C 90.000,E1 274.531} C_DIS
LIN {X 0.124,Y -489.735,Z 975.522,A 0.000,B 0.000,C 90.000,E1 274.012} C_DIS
LIN {X -0.177,Y -488.579,Z 975.520,A 0.000,B 0.000,C 90.000,E1 273.555} C_DIS
LIN {X 0.037,Y -486.909,Z 975.517,A 0.000,B 0.000,C 90.000,E1 273.037} C_DIS
LIN {X 0.217,Y -484.581,Z 975.514,A 0.000,B 0.000,C 90.000,E1 272.522} C_DIS
LIN {X -0.098,Y -481.506,Z 975.511,A 0.000,B 0.000,C 90.000,E1 272.064} C_DIS
LIN {X 0.068,Y -477.590,Z 975.509,A 0.000,B 0.000,C 90.000,E1 271.547} C_DIS
LIN {X 0.197,Y -472.657,Z 975.506,A 0.000,B 0.000,C 90.000,E1 271.031} C_DIS
LIN {X 0.002,Y -466.817,Z 975.503,A 0.000,B 0.000,C 90.000,E1 270.573} C_DIS
LIN {X -0.173,Y -460.622,Z 975.501,A 0.000,B 0.000,C 90.000,E1 270.172} C_DIS
LIN {X 0.079,Y -453.991,Z 975.499,A 0.000,B 0.000,C 90.000,E1 269.771} C_DIS
LIN {X -0.147,Y -447.130,Z 975.497,A 0.000,B 0.000,C 90.000,E1 269.484} C_DIS
LIN {X 0.031,Y -439.869,Z 975.496,A 0.000,B 0.000,C 90.000,E1 269.198} C_DIS
LIN {X 0.150,Y -432.117,Z 975.494,A 0.000,B 0.000,C 90.000,E1 268.969} C_DIS
LIN {X -0.210,Y -424.410,Z 975.493,A 0.000,B 0.000,C 90.000,E1 268.854} C_DIS
LIN {X 0.120,Y -416.314,Z 975.493,A 0.000,B 0.000,C 90.000,E1 268.682} C_DIS
LIN {X -0.171,Y -404.798,Z 975.492,A 0.000,B 0.000,C 90.000,E1 268.625} C_DIS
LIN {X 0.174,Y -402.436,Z 975.492,A 0.000,B 0.000,C 90.000,E1 268.568} C_DIS
LIN {X 0.052,Y -181.230,Z 975.492,A 0.000,B 0.000,C 90.000,E1 268.568} C_DIS
LIN {X -0.047,Y -180.891,Z 975.473,A 0.000,B 0.000,C 90.000,E1 265.179} C_DIS
LIN {X 0.015,Y -179.017,Z 975.445,A 0.000,B 0.000,C 90.000,E1 260.095} C_DIS
LIN {X -0.065,Y -178.644,Z 975.440,A 0.000,B 0.000,C 90.000,E1 259.275} C_DIS
LIN {X 0.008,Y -175.695,Z 975.412,A 0.000,B 0.000,C 90.000,E1 254.157} C_DIS
LIN {X 0.018,Y -172.412,Z 975.388,A 0.000,B 0.000,C 90.000,E1 249.880} C_DIS
LIN {X 0.035,Y -171.227,Z 975.379,A 0.000,B 0.000,C 90.000,E1 248.156} C_DIS
LIN {X 0.010,Y -167.508,Z 975.355,A 0.000,B 0.000,C 90.000,E1 243.845} C_DIS
LIN {X -0.057,Y -166.904,Z 975.350,A 0.000,B 0.000,C 90.000,E1 242.999} C_DIS
LIN {X -0.005,Y -162.211,Z 975.321,A 0.000,B 0.000,C 90.000,E1 237.740} C_DIS
LIN {X 0.049,Y -160.788,Z 975.311,A 0.000,B 0.000,C 90.000,E1 235.960} C_DIS
LIN {X 0.020,Y -157.579,Z 975.291,A 0.000,B 0.000,C 90.000,E1 232.431} C_DIS
LIN {X 0.053,Y -155.611,Z 975.276,A 0.000,B 0.000,C 90.000,E1 229.747} C_DIS
LIN {X -0.003,Y -151.890,Z 975.252,A 0.000,B 0.000,C 90.000,E1 225.283} C_DIS
LIN {X -0.095,Y -150.118,Z 975.237,A 0.000,B 0.000,C 90.000,E1 222.609} C_DIS
LIN {X 0.033,Y -146.911,Z 975.211,A 0.000,B 0.000,C 90.000,E1 218.016} C_DIS
LIN {X -0.066,Y -145.498,Z 975.196,A 0.000,B 0.000,C 90.000,E1 215.311} C_DIS
LIN {X 0.053,Y -142.903,Z 975.170,A 0.000,B 0.000,C 90.000,E1 210.669} C_DIS
LIN {X -0.017,Y -141.523,Z 975.150,A 0.000,B 0.000,C 90.000,E1 207.001} C_DIS
LIN {X 0.027,Y -139.396,Z 975.114,A 0.000,B 0.000,C 90.000,E1 200.482} C_DIS
LIN {X 0.078,Y -139.108,Z 975.104,A 0.000,B 0.000,C 90.000,E1 198.598} C_DIS
LIN {X -0.067,Y -138.353,Z 975.057,A 0.000,B 0.000,C 90.000,E1 190.254} C_DIS
LIN {X 0.063,Y -139.510,Z 975.005,A 0.000,B 0.000,C 90.000,E1 180.859} C_DIS
LIN {X 0.003,Y -141.152,Z 974.974,A 0.000,B 0.000,C 90.000,E1 175.298} C_DIS
LIN {X -0.026,Y -142.532,Z 974.958,A 0.000,B 0.000,C 90.000,E1 172.527} C_DIS
LIN {X 0.042,Y -144.800,Z 974.933,A 0.000,B 0.000,C 90.000,E1 167.881} C_DIS
LIN {X 0.031,Y -147.419,Z 974.912,A 0.000,B 0.000,C 90.000,E1 164.212} C_DIS
LIN {X 0.060,Y -149.996,Z 974.892,A 0.000,B 0.000,C 90.000,E1 160.550} C_DIS
LIN {X 0.067,Y -153.324,Z 974.872,A 0.000,B 0.000,C 90.000,E1 156.922} C_DIS
LIN {X -0.021,Y -155.024,Z 974.862,A 0.000,B 0.000,C 90.000,E1 155.153} C_DIS
LIN {X 0.000,Y -158.671,Z 974.842,A 0.000,B 0.000,C 90.000,E1 151.563} C_DIS
LIN {X 0.083,Y -161.950,Z 974.827,A 0.000,B 0.000,C 90.000,E1 148.869} C_DIS
LIN {X -0.032,Y -166.141,Z 974.808,A 0.000,B 0.000,C 90.000,E1 145.388} C_DIS
LIN {X -0.036,Y -171.153,Z 974.788,A 0.000,B 0.000,C 90.000,E1 141.904} C_DIS
LIN {X -0.001,Y -176.032,Z 974.769,A 0.000,B 0.000,C 90.000,E1 138.447} C_DIS
LIN {X -0.006,Y -180.284,Z 974.755,A 0.000,B 0.000,C 90.000,E1 135.891} C_DIS
LIN {X -0.034,Y -185.697,Z 974.736,A 0.000,B 0.000,C 90.000,E1 132.528} C_DIS
LIN {X 0.019,Y -190.302,Z 974.722,A 0.000,B 0.000,C 90.000,E1 130.011} C_DIS
LIN {X -0.023,Y -195.268,Z 974.706,A 0.000,B 0.000,C 90.000,E1 127.156} C_DIS
LIN {X -0.068,Y -298.243,Z 974.706,A 0.000,B 0.000,C 90.000,E1 127.156} C_DIS
LIN {X 0.112,Y -301.030,Z 974.706,A 0.000,B 0.000,C 90.000,E1 127.076} C_DIS
LIN {X -0.035,Y -304.892,Z 974.705,A 0.000,B 0.000,C 90.000,E1 126.916} C_DIS
LIN {X 0.060,Y -307.189,Z 974.704,A 0.000,B 0.000,C 90.000,E1 126.710} C_DIS
LIN {X 0.127,Y -311.049,Z 974.701,A 0.000,B 0.000,C 90.000,E1 126.217} C_DIS
LIN {X -0.091,Y -312.869,Z 974.700,A 0.000,B 0.000,C 90.000,E1 125.931} C_DIS
LIN {X -0.057,Y -314.291,Z 974.698,A 0.000,B 0.000,C 90.000,E1 125.598} C_DIS
LIN {X -0.129,Y -326.054,Z 974.678,A 0.000,B 0.000,C 90.000,E1 122.084} C_DIS
LIN {X 0.159,Y -337.005,Z 974.662,A 0.000,B 0.000,C 90.000,E1 119.205} C_DIS
LIN {X -0.193,Y -349.344,Z 974.647,A 0.000,B 0.000,C 90.000,E1 116.488} C_DIS
LIN {X -0.202,Y -363.184,Z 974.632,A 0.000,B 0.000,C 90.000,E1 113.770} C_DIS
LIN {X 0.138,Y -376.842,Z 974.619,A 0.000,B 0.000,C 90.000,E1 111.354} C_DIS
LIN {X -0.157,Y -391.878,Z 974.606,A 0.000,B 0.000,C 90.000,E1 109.087} C_DIS
LIN {X 0.031,Y -408.398,Z 974.593,A 0.000,B 0.000,C 90.000,E1 106.804} C_DIS
LIN {X 0.126,Y -426.522,Z 974.581,A 0.000,B 0.000,C 90.000,E1 104.592} C_DIS
LIN {X 0.082,Y -446.182,Z 974.569,A 0.000,B 0.000,C 90.000,E1 102.479} C_DIS
LIN {X -0.081,Y -466.521,Z 974.559,A 0.000,B 0.000,C 90.000,E1 100.546} C_DIS
LIN {X -0.047,Y -468.737,Z 974.557,A 0.000,B 0.000,C 90.000,E1 100.310} C_DIS
LIN {X -0.012,Y -470.411,Z 974.556,A 0.000,B 0.000,C 90.000,E1 100.074} C_DIS
LIN {X -0.242,Y -471.808,Z 974.555,A 0.000,B 0.000,C 90.000,E1 99.849} C_DIS
LIN {X 0.075,Y -472.846,Z 974.553,A 0.000,B 0.000,C 90.000,E1 99.557} C_DIS
LIN {X 0.259,Y -474.049,Z 974.550,A 0.000,B 0.000,C 90.000,E1 99.029} C_DIS
LIN {X -0.095,Y -474.249,Z 974.548,A 0.000,B 0.000,C 90.000,E1 98.568} C_DIS
LIN {X 0.030,Y -473.484,Z 974.545,A 0.000,B 0.000,C 90.000,E1 98.049} C_DIS
LIN {X 0.157,Y -471.629,Z 974.542,A 0.000,B 0.000,C 90.000,E1 97.530} C_DIS
LIN {X 0.013,Y -470.184,Z 974.541,A 0.000,B 0.000,C 90.000,E1 97.296} C_DIS
LIN {X -0.117,Y -456.657,Z 974.529,A 0.000,B 0.000,C 90.000,E1 95.277} C_DIS
LIN {X 0.081,Y -444.678,Z 974.519,A 0.000,B 0.000,C 90.000,E1 93.440} C_DIS
LIN {X 0.182,Y -426.499,Z 974.503,A 0.000,B 0.000,C 90.000,E1 90.516} C_DIS
LIN {X 0.047,Y -411.404,Z 974.488,A 0.000,B 0.000,C 90.000,E1 87.822} C_DIS
LIN {X 0.087,Y -402.395,Z 974.479,A 0.000,B 0.000,C 90.000,E1 86.159} C_DIS
LIN {X 0.044,Y -391.694,Z 974.468,A 0.000,B 0.000,C 90.000,E1 84.204} C_DIS
LIN {X -0.158,Y -382.322,Z 974.458,A 0.000,B 0.000,C 90.000,E1 82.527} C_DIS
LIN {X -0.142,Y -372.746,Z 974.449,A 0.000,B 0.000,C 90.000,E1 80.792} C_DIS
LIN {X 0.111,Y -362.852,Z 974.439,A 0.000,B 0.000,C 90.000,E1 78.993} C_DIS
LIN {X -0.035,Y -352.734,Z 974.429,A 0.000,B 0.000,C 90.000,E1 77.229} C_DIS
LIN {X 0.007,Y -334.739,Z 974.410,A 0.000,B 0.000,C 90.000,E1 73.866} C_DIS
LIN {X 0.085,Y -322.421,Z 974.396,A 0.000,B 0.000,C 90.000,E1 71.348} C_DIS
LIN {X -0.037,Y -311.808,Z 974.384,A 0.000,B 0.000,C 90.000,E1 69.135} C_DIS
LIN {X -0.079,Y -299.867,Z 974.370,A 0.000,B 0.000,C 90.000,E1 66.538} C_DIS
LIN {X 0.082,Y -288.102,Z 974.355,A 0.000,B 0.000,C 90.000,E1 63.845} C_DIS
LIN {X -0.140,Y -277.854,Z 974.342,A 0.000,B 0.000,C 90.000,E1 61.513} C_DIS
LIN {X 0.151,Y -264.971,Z 974.324,A 0.000,B 0.000,C 90.000,E1 58.329} C_DIS
LIN {X 0.024,Y -253.912,Z 974.308,A 0.000,B 0.000,C 90.000,E1 55.515} C_DIS
LIN {X -0.085,Y -242.079,Z 974.290,A 0.000,B 0.000,C 90.000,E1 52.271} C_DIS
LIN {X -0.113,Y -231.136,Z 974.272,A 0.000,B 0.000,C 90.000,E1 48.933} C_DIS
LIN {X -0.011,Y -220.918,Z 974.253,A 0.000,B 0.000,C 90.000,E1 45.486} C_DIS
LIN {X -0.016,Y -211.392,Z 974.233,A 0.000,B 0.000,C 90.000,E1 42.000} C_DIS
LIN {X 0.029,Y -203.505,Z 974.216,A 0.000,B 0.000,C 90.000,E1 38.830} C_DIS
LIN {X 0.098,Y -196.281,Z 974.198,A 0.000,B 0.000,C 90.000,E1 35.598} C_DIS
LIN {X 0.080,Y -189.713,Z 974.180,A 0.000,B 0.000,C 90.000,E1 32.339} C_DIS
LIN {X -0.077,Y -183.876,Z 974.161,A 0.000,B 0.000,C 90.000,E1 29.077} C_DIS
LIN {X -0.064,Y -178.760,Z 974.143,A 0.000,B 0.000,C 90.000,E1 25.720} C_DIS
LIN {X -0.083,Y -174.406,Z 974.124,A 0.000,B 0.000,C 90.000,E1 22.333} C_DIS
LIN {X -0.079,Y -170.734,Z 974.105,A 0.000,B 0.000,C 90.000,E1 18.906} C_DIS
LIN {X 0.057,Y -167.125,Z 974.081,A 0.000,B 0.000,C 90.000,E1 14.537} C_DIS
LIN {X 0.004,Y -164.171,Z 974.052,A 0.000,B 0.000,C 90.000,E1 9.321} C_DIS
LIN {X 0.000,Y -162.538,Z 974.000,A 0.000,B 0.000,C 90.000,E1 360.000} C_DIS
LIN {X 0.081,Y -164.475,Z 973.958,A 0.000,B 0.000,C 90.000,E1 352.470} C_DIS
LIN {X 0.064,Y -167.669,Z 973.929,A 0.000,B 0.000,C 90.000,E1 347.229} C_DIS
LIN {X -0.055,Y -170.715,Z 973.910,A 0.000,B 0.000,C 90.000,E1 343.795} C_DIS
LIN {X 0.036,Y -174.477,Z 973.891,A 0.000,B 0.000,C 90.000,E1 340.315} C_DIS
LIN {X -0.039,Y -179.031,Z 973.872,A 0.000,B 0.000,C 90.000,E1 336.922} C_DIS
LIN {X 0.051,Y -184.364,Z 973.853,A 0.000,B 0.000,C 90.000,E1 333.512} C_DIS
LIN {X -0.058,Y -190.379,Z 973.834,A 0.000,B 0.000,C 90.000,E1 330.205} C_DIS
LIN {X -0.067,Y -197.067,Z 973.816,A 0.000,B 0.000,C 90.000,E1 326.914} C_DIS
LIN {X 0.095,Y -204.222,Z 973.798,A 0.000,B 0.000,C 90.000,E1 323.623} C_DIS
LIN {X 0.072,Y -211.992,Z 973.780,A 0.000,B 0.000,C 90.000,E1 320.436} C_DIS
LIN {X -0.040,Y -221.308,Z 973.761,A 0.000,B 0.000,C 90.000,E1 316.944} C_DIS
LIN {X -0.009,Y -230.574,Z 973.744,A 0.000,B 0.000,C 90.000,E1 313.866} C_DIS
LIN {X -0.108,Y -237.129,Z 973.733,A 0.000,B 0.000,C 90.000,E1 312.000} C_DIS
LIN {X 0.069,Y -245.965,Z 973.721,A 0.000,B 0.000,C 90.000,E1 309.725} C_DIS
LIN {X 0.095,Y -254.181,Z 973.711,A 0.000,B 0.000,C 90.000,E1 307.890} C_DIS
LIN {X 0.038,Y -267.048,Z 973.697,A 0.000,B 0.000,C 90.000,E1 305.391} C_DIS
LIN {X -0.039,Y -281.089,Z 973.683,A 0.000,B 0.000,C 90.000,E1 302.959} C_DIS
LIN {X -0.127,Y -298.351,Z 973.668,A 0.000,B 0.000,C 90.000,E1 300.256} C_DIS
LIN {X 0.139,Y -314.561,Z 973.655,A 0.000,B 0.000,C 90.000,E1 297.897} C_DIS
LIN {X 0.178,Y -329.942,Z 973.644,A 0.000,B 0.000,C 90.000,E1 295.976} C_DIS
LIN {X -0.006,Y -356.234,Z 973.629,A 0.000,B 0.000,C 90.000,E1 293.153} C_DIS
LIN {X -0.108,Y -372.541,Z 973.620,A 0.000,B 0.000,C 90.000,E1 291.535} C_DIS
LIN {X 0.122,Y -388.721,Z 973.611,A 0.000,B 0.000,C 90.000,E1 289.939} C_DIS
LIN {X -0.170,Y -399.334,Z 973.605,A 0.000,B 0.000,C 90.000,E1 288.960} C_DIS
LIN {X 0.169,Y -409.720,Z 973.599,A 0.000,B 0.000,C 90.000,E1 287.873} C_DIS
LIN {X -0.156,Y -419.828,Z 973.594,A 0.000,B 0.000,C 90.000,E1 286.858} C_DIS
LIN {X -0.254,Y -429.587,Z 973.588,A 0.000,B 0.000,C 90.000,E1 285.788} C_DIS
LIN {X 0.151,Y -438.821,Z 973.582,A 0.000,B 0.000,C 90.000,E1 284.662} C_DIS
LIN {X -0.187,Y -447.409,Z 973.576,A 0.000,B 0.000,C 90.000,E1 283.647} C_DIS
LIN {X -0.103,Y -455.518,Z 973.570,A 0.000,B 0.000,C 90.000,E1 282.591} C_DIS
LIN {X 0.081,Y -463.212,Z 973.564,A 0.000,B 0.000,C 90.000,E1 281.535} C_DIS
LIN {X -0.193,Y -470.368,Z 973.558,A 0.000,B 0.000,C 90.000,E1 280.546} C_DIS
LIN {X -0.165,Y -475.219,Z 973.554,A 0.000,B 0.000,C 90.000,E1 279.782} C_DIS
LIN {X -0.184,Y -479.421,Z 973.550,A 0.000,B 0.000,C 90.000,E1 279.029} C_DIS
LIN {X -0.159,Y -482.961,Z 973.546,A 0.000,B 0.000,C 90.000,E1 278.276} C_DIS
LIN {X -0.171,Y -485.910,Z 973.542,A 0.000,B 0.000,C 90.000,E1 277.530} C_DIS
LIN {X 0.078,Y -487.512,Z 973.539,A 0.000,B 0.000,C 90.000,E1 277.004} C_DIS
LIN {X -0.211,Y -488.800,Z 973.536,A 0.000,B 0.000,C 90.000,E1 276.543} C_DIS
LIN {X -0.056,Y -489.738,Z 973.533,A 0.000,B 0.000,C 90.000,E1 276.030} C_DIS
LIN {X 0.163,Y -490.344,Z 973.531,A 0.000,B 0.000,C 90.000,E1 275.511} C_DIS
LIN {X -0.104,Y -490.595,Z 973.528,A 0.000,B 0.000,C 90.000,E1 275.049} C_DIS
LIN {X 0.121,Y -490.414,Z 973.525,A 0.000,B 0.000,C 90.000,E1 274.531} C_DIS
LIN {X -0.146,Y -489.859,Z 973.523,A 0.000,B 0.000,C 90.000,E1 274.069} C_DIS
LIN {X 0.042,Y -488.760,Z 973.520,A 0.000,B 0.000,C 90.000,E1 273.555} C_DIS
LIN {X -0.230,Y -487.130,Z 973.517,A 0.000,B 0.000,C 90.000,E1 273.094} C_DIS
LIN {X -0.049,Y -484.830,Z 973.514,A 0.000,B 0.000,C 90.000,E1 272.579} C_DIS
LIN {X 0.119,Y -481.810,Z 973.512,A 0.000,B 0.000,C 90.000,E1 272.064} C_DIS
LIN {X -0.044,Y -480.051,Z 973.510,A 0.000,B 0.000,C 90.000,E1 271.835} C_DIS
LIN {X 0.113,Y -475.647,Z 973.507,A 0.000,B 0.000,C 90.000,E1 271.318} C_DIS
LIN {X -0.058,Y -473.122,Z 973.506,A 0.000,B 0.000,C 90.000,E1 271.088} C_DIS
LIN {X 0.155,Y -467.225,Z 973.503,A 0.000,B 0.000,C 90.000,E1 270.573} C_DIS
LIN {X -0.050,Y -461.059,Z 973.501,A 0.000,B 0.000,C 90.000,E1 270.172} C_DIS
LIN {X 0.188,Y -454.549,Z 973.499,A 0.000,B 0.000,C 90.000,E1 269.771} C_DIS
LIN {X -0.067,Y -447.726,Z 973.497,A 0.000,B 0.000,C 90.000,E1 269.484} C_DIS
LIN {X 0.066,Y -440.402,Z 973.496,A 0.000,B 0.000,C 90.000,E1 269.198} C_DIS
LIN {X 0.170,Y -432.828,Z 973.494,A 0.000,B 0.000,C 90.000,E1 268.969} C_DIS
LIN {X -0.213,Y -425.247,Z 973.493,A 0.000,B 0.000,C 90.000,E1 268.854} C_DIS
LIN {X 0.097,Y -417.422,Z 973.493,A 0.000,B 0.000,C 90.000,E1 268.682} C_DIS
LIN {X 0.178,Y -406.700,Z 973.492,A 0.000,B 0.000,C 90.000,E1 268.568} C_DIS
LIN {X 0.056,Y -403.026,Z 973.492,A 0.000,B 0.000,C 90.000,E1 268.568} C_DIS
LIN {X -0.003,Y -181.227,Z 973.492,A 0.000,B 0.000,C 90.000,E1 268.568} C_DIS
LIN {X -0.080,Y -180.890,Z 973.473,A 0.000,B 0.000,C 90.000,E1 265.179} C_DIS
LIN {X -0.018,Y -179.014,Z 973.445,A 0.000,B 0.000,C 90.000,E1 260.095} C_DIS
LIN {X 0.077,Y -178.637,Z 973.440,A 0.000,B 0.000,C 90.000,E1 259.218} C_DIS
LIN {X -0.025,Y -175.688,Z 973.412,A 0.000,B 0.000,C 90.000,E1 254.157} C_DIS
LIN {X -0.014,Y -172.404,Z 973.388,A 0.000,B 0.000,C 90.000,E1 249.880} C_DIS
LIN {X 0.002,Y -171.216,Z 973.379,A 0.000,B 0.000,C 90.000,E1 248.156} C_DIS
LIN {X -0.021,Y -167.500,Z 973.355,A 0.000,B 0.000,C 90.000,E1 243.845} C_DIS
LIN {X -0.088,Y -166.896,Z 973.350,A 0.000,B 0.000,C 90.000,E1 242.999} C_DIS
LIN {X -0.035,Y -162.203,Z 973.321,A 0.000,B 0.000,C 90.000,E1 237.740} C_DIS
LIN {X 0.018,Y -160.777,Z 973.311,A 0.000,B 0.000,C 90.000,E1 235.960} C_DIS
LIN {X -0.010,Y -157.570,Z 973.291,A 0.000,B 0.000,C 90.000,E1 232.431} C_DIS
LIN {X 0.023,Y -155.601,Z 973.276,A 0.000,B 0.000,C 90.000,E1 229.747} C_DIS
LIN {X 0.075,Y -151.882,Z 973.252,A 0.000,B 0.000,C 90.000,E1 225.243} C_DIS
LIN {X 0.088,Y -150.109,Z 973.236,A 0.000,B 0.000,C 90.000,E1 222.528} C_DIS
LIN {X 0.005,Y -146.903,Z 973.211,A 0.000,B 0.000,C 90.000,E1 218.016} C_DIS
LIN {X 0.025,Y -145.492,Z 973.196,A 0.000,B 0.000,C 90.000,E1 215.264} C_DIS
LIN {X 0.025,Y -142.898,Z 973.170,A 0.000,B 0.000,C 90.000,E1 210.669} C_DIS
LIN {X -0.045,Y -141.518,Z 973.150,A 0.000,B 0.000,C 90.000,E1 207.001} C_DIS
LIN {X -0.002,Y -139.394,Z 973.114,A 0.000,B 0.000,C 90.000,E1 200.482} C_DIS
LIN {X 0.049,Y -139.105,Z 973.103,A 0.000,B 0.000,C 90.000,E1 198.598} C_DIS
LIN {X 0.041,Y -138.353,Z 973.057,A 0.000,B 0.000,C 90.000,E1 190.197} C_DIS
LIN {X 0.035,Y -139.511,Z 973.005,A 0.000,B 0.000,C 90.000,E1 180.859} C_DIS
LIN {X -0.025,Y -141.157,Z 972.974,A 0.000,B 0.000,C 90.000,E1 175.298} C_DIS
LIN {X -0.054,Y -142.537,Z 972.958,A 0.000,B 0.000,C 90.000,E1 172.527} C_DIS
LIN {X 0.014,Y -144.807,Z 972.933,A 0.000,B 0.000,C 90.000,E1 167.881} C_DIS
LIN {X 0.002,Y -147.427,Z 972.912,A 0.000,B 0.000,C 90.000,E1 164.212} C_DIS
LIN {X 0.030,Y -150.005,Z 972.892,A 0.000,B 0.000,C 90.000,E1 160.550} C_DIS
LIN {X 0.038,Y -153.336,Z 972.872,A 0.000,B 0.000,C 90.000,E1 156.922} C_DIS
LIN {X 0.019,Y -155.871,Z 972.857,A 0.000,B 0.000,C 90.000,E1 154.229} C_DIS
LIN {X -0.015,Y -159.725,Z 972.837,A 0.000,B 0.000,C 90.000,E1 150.667} C_DIS
LIN {X 0.052,Y -161.964,Z 972.827,A 0.000,B 0.000,C 90.000,E1 148.869} C_DIS
LIN {X -0.064,Y -166.155,Z 972.808,A 0.000,B 0.000,C 90.000,E1 145.388} C_DIS
LIN {X -0.069,Y -171.168,Z 972.788,A 0.000,B 0.000,C 90.000,E1 141.904} C_DIS
LIN {X -0.035,Y -176.048,Z 972.769,A 0.000,B 0.000,C 90.000,E1 138.447} C_DIS
LIN {X -0.039,Y -180.304,Z 972.755,A 0.000,B 0.000,C 90.000,E1 135.891} C_DIS
LIN {X -0.067,Y -185.715,Z 972.736,A 0.000,B 0.000,C 90.000,E1 132.528} C_DIS
LIN {X -0.016,Y -190.322,Z 972.722,A 0.000,B 0.000,C 90.000,E1 130.011} C_DIS
LIN {X 0.078,Y -195.213,Z 972.707,A 0.000,B 0.000,C 90.000,E1 127.156} C_DIS
LIN {X 0.083,Y -298.856,Z 972.707,A 0.000,B 0.000,C 90.000,E1 127.156} C_DIS
LIN {X -0.084,Y -300.605,Z 972.706,A 0.000,B 0.000,C 90.000,E1 127.156} C_DIS
LIN {X -0.131,Y -305.029,Z 972.705,A 0.000,B 0.000,C 90.000,E1 126.950} C_DIS
LIN {X 0.006,Y -307.520,Z 972.704,A 0.000,B 0.000,C 90.000,E1 126.710} C_DIS
LIN {X -0.039,Y -311.329,Z 972.701,A 0.000,B 0.000,C 90.000,E1 126.217} C_DIS
LIN {X -0.004,Y -313.056,Z 972.699,A 0.000,B 0.000,C 90.000,E1 125.884} C_DIS
LIN {X -0.040,Y -314.410,Z 972.698,A 0.000,B 0.000,C 90.000,E1 125.564} C_DIS
LIN {X 0.152,Y -326.139,Z 972.678,A 0.000,B 0.000,C 90.000,E1 122.005} C_DIS
LIN {X -0.013,Y -337.105,Z 972.662,A 0.000,B 0.000,C 90.000,E1 119.205} C_DIS
LIN {X -0.056,Y -349.459,Z 972.647,A 0.000,B 0.000,C 90.000,E1 116.437} C_DIS
LIN {X 0.098,Y -363.315,Z 972.632,A 0.000,B 0.000,C 90.000,E1 113.695} C_DIS
LIN {X -0.044,Y -376.988,Z 972.619,A 0.000,B 0.000,C 90.000,E1 111.354} C_DIS
LIN {X 0.028,Y -392.040,Z 972.606,A 0.000,B 0.000,C 90.000,E1 109.033} C_DIS
LIN {X -0.158,Y -408.578,Z 972.593,A 0.000,B 0.000,C 90.000,E1 106.804} C_DIS
LIN {X -0.068,Y -426.722,Z 972.581,A 0.000,B 0.000,C 90.000,E1 104.592} C_DIS
LIN {X -0.111,Y -446.395,Z 972.569,A 0.000,B 0.000,C 90.000,E1 102.479} C_DIS
LIN {X 0.192,Y -466.741,Z 972.558,A 0.000,B 0.000,C 90.000,E1 100.489} C_DIS
LIN {X 0.202,Y -468.929,Z 972.557,A 0.000,B 0.000,C 90.000,E1 100.254} C_DIS
LIN {X 0.211,Y -470.581,Z 972.556,A 0.000,B 0.000,C 90.000,E1 100.018} C_DIS
LIN {X -0.017,Y -471.939,Z 972.554,A 0.000,B 0.000,C 90.000,E1 99.792} C_DIS
LIN {X -0.165,Y -472.944,Z 972.553,A 0.000,B 0.000,C 90.000,E1 99.557} C_DIS
LIN {X 0.019,Y -474.093,Z 972.550,A 0.000,B 0.000,C 90.000,E1 99.029} C_DIS
LIN {X 0.135,Y -474.247,Z 972.547,A 0.000,B 0.000,C 90.000,E1 98.511} C_DIS
LIN {X -0.209,Y -473.431,Z 972.545,A 0.000,B 0.000,C 90.000,E1 98.049} C_DIS
LIN {X -0.081,Y -471.514,Z 972.542,A 0.000,B 0.000,C 90.000,E1 97.530} C_DIS
LIN {X 0.099,Y -468.307,Z 972.539,A 0.000,B 0.000,C 90.000,E1 97.004} C_DIS
LIN {X -0.123,Y -454.818,Z 972.528,A 0.000,B 0.000,C 90.000,E1 94.992} C_DIS
LIN {X -0.190,Y -441.176,Z 972.516,A 0.000,B 0.000,C 90.000,E1 92.922} C_DIS
LIN {X -0.042,Y -426.404,Z 972.503,A 0.000,B 0.000,C 90.000,E1 90.516} C_DIS
LIN {X -0.172,Y -411.288,Z 972.488,A 0.000,B 0.000,C 90.000,E1 87.822} C_DIS
LIN {X -0.130,Y -402.249,Z 972.479,A 0.000,B 0.000,C 90.000,E1 86.159} C_DIS
LIN {X -0.170,Y -391.557,Z 972.468,A 0.000,B 0.000,C 90.000,E1 84.204} C_DIS
LIN {X 0.010,Y -382.197,Z 972.458,A 0.000,B 0.000,C 90.000,E1 82.470} C_DIS
LIN {X 0.008,Y -374.223,Z 972.450,A 0.000,B 0.000,C 90.000,E1 81.027} C_DIS
LIN {X -0.077,Y -364.394,Z 972.440,A 0.000,B 0.000,C 90.000,E1 79.285} C_DIS
LIN {X 0.107,Y -352.599,Z 972.429,A 0.000,B 0.000,C 90.000,E1 77.173} C_DIS
LIN {X -0.097,Y -334.580,Z 972.410,A 0.000,B 0.000,C 90.000,E1 73.850} C_DIS
LIN {X -0.154,Y -320.768,Z 972.395,A 0.000,B 0.000,C 90.000,E1 71.040} C_DIS
LIN {X -0.014,Y -310.152,Z 972.382,A 0.000,B 0.000,C 90.000,E1 68.773} C_DIS
LIN {X -0.103,Y -298.238,Z 972.368,A 0.000,B 0.000,C 90.000,E1 66.177} C_DIS
LIN {X -0.121,Y -286.499,Z 972.353,A 0.000,B 0.000,C 90.000,E1 63.512} C_DIS
LIN {X -0.119,Y -276.228,Z 972.339,A 0.000,B 0.000,C 90.000,E1 61.129} C_DIS
LIN {X -0.024,Y -264.794,Z 972.324,A 0.000,B 0.000,C 90.000,E1 58.329} C_DIS
LIN {X 0.061,Y -253.760,Z 972.308,A 0.000,B 0.000,C 90.000,E1 55.468} C_DIS
LIN {X 0.086,Y -241.924,Z 972.290,A 0.000,B 0.000,C 90.000,E1 52.190} C_DIS
LIN {X 0.048,Y -231.014,Z 972.271,A 0.000,B 0.000,C 90.000,E1 48.852} C_DIS
LIN {X -0.015,Y -220.818,Z 972.252,A 0.000,B 0.000,C 90.000,E1 45.445} C_DIS
LIN {X -0.031,Y -211.340,Z 972.233,A 0.000,B 0.000,C 90.000,E1 41.962} C_DIS
LIN {X -0.123,Y -203.475,Z 972.216,A 0.000,B 0.000,C 90.000,E1 38.830} C_DIS
LIN {X -0.049,Y -196.264,Z 972.198,A 0.000,B 0.000,C 90.000,E1 35.598} C_DIS
LIN {X -0.063,Y -189.723,Z 972.180,A 0.000,B 0.000,C 90.000,E1 32.339} C_DIS
LIN {X 0.036,Y -183.905,Z 972.161,A 0.000,B 0.000,C 90.000,E1 28.999} C_DIS
LIN {X -0.036,Y -178.804,Z 972.143,A 0.000,B 0.000,C 90.000,E1 25.668} C_DIS
LIN {X -0.050,Y -174.466,Z 972.124,A 0.000,B 0.000,C 90.000,E1 22.280} C_DIS
LIN {X -0.042,Y -170.799,Z 972.105,A 0.000,B 0.000,C 90.000,E1 18.852} C_DIS
LIN {X -0.064,Y -167.200,Z 972.081,A 0.000,B 0.000,C 90.000,E1 14.537} C_DIS
LIN {X 0.051,Y -164.247,Z 972.052,A 0.000,B 0.000,C 90.000,E1 9.265} C_DIS
LIN {X -0.029,Y -162.696,Z 971.997,A 0.000,B 0.000,C 90.000,E1 359.542} C_DIS
LIN {X 0.087,Y -164.609,Z 971.958,A 0.000,B 0.000,C 90.000,E1 352.470} C_DIS
LIN {X 0.076,Y -167.815,Z 971.929,A 0.000,B 0.000,C 90.000,E1 347.229} C_DIS
LIN {X -0.041,Y -170.880,Z 971.910,A 0.000,B 0.000,C 90.000,E1 343.795} C_DIS
LIN {X 0.056,Y -174.635,Z 971.891,A 0.000,B 0.000,C 90.000,E1 340.315} C_DIS
LIN {X -0.015,Y -179.200,Z 971.872,A 0.000,B 0.000,C 90.000,E1 336.922} C_DIS
LIN {X 0.081,Y -184.538,Z 971.853,A 0.000,B 0.000,C 90.000,E1 333.512} C_DIS
LIN {X -0.022,Y -190.558,Z 971.834,A 0.000,B 0.000,C 90.000,E1 330.205} C_DIS
LIN {X -0.026,Y -197.217,Z 971.816,A 0.000,B 0.000,C 90.000,E1 326.914} C_DIS
LIN {X 0.020,Y -204.393,Z 971.798,A 0.000,B 0.000,C 90.000,E1 323.657} C_DIS
LIN {X 0.024,Y -213.159,Z 971.778,A 0.000,B 0.000,C 90.000,E1 320.070} C_DIS
LIN {X 0.094,Y -222.579,Z 971.759,A 0.000,B 0.000,C 90.000,E1 316.539} C_DIS
LIN {X 0.005,Y -232.025,Z 971.742,A 0.000,B 0.000,C 90.000,E1 313.500} C_DIS
LIN {X 0.097,Y -238.720,Z 971.731,A 0.000,B 0.000,C 90.000,E1 311.595} C_DIS
LIN {X -0.039,Y -247.692,Z 971.719,A 0.000,B 0.000,C 90.000,E1 309.402} C_DIS
LIN {X 0.001,Y -256.035,Z 971.709,A 0.000,B 0.000,C 90.000,E1 307.569} C_DIS
LIN {X 0.107,Y -271.013,Z 971.693,A 0.000,B 0.000,C 90.000,E1 304.692} C_DIS
LIN {X 0.050,Y -289.611,Z 971.676,A 0.000,B 0.000,C 90.000,E1 301.592} C_DIS
LIN {X -0.098,Y -309.717,Z 971.659,A 0.000,B 0.000,C 90.000,E1 298.615} C_DIS
LIN {X -0.143,Y -322.031,Z 971.650,A 0.000,B 0.000,C 90.000,E1 297.001} C_DIS
LIN {X 0.128,Y -337.952,Z 971.639,A 0.000,B 0.000,C 90.000,E1 295.079} C_DIS
LIN {X 0.113,Y -362.381,Z 971.625,A 0.000,B 0.000,C 90.000,E1 292.514} C_DIS
LIN {X 0.118,Y -381.062,Z 971.615,A 0.000,B 0.000,C 90.000,E1 290.663} C_DIS
LIN {X 0.189,Y -396.818,Z 971.607,A 0.000,B 0.000,C 90.000,E1 289.141} C_DIS
LIN {X 0.057,Y -407.241,Z 971.601,A 0.000,B 0.000,C 90.000,E1 288.127} C_DIS
LIN {X -0.097,Y -417.415,Z 971.595,A 0.000,B 0.000,C 90.000,E1 287.094} C_DIS
LIN {X -0.136,Y -427.190,Z 971.589,A 0.000,B 0.000,C 90.000,E1 286.024} C_DIS
LIN {X -0.137,Y -436.511,Z 971.583,A 0.000,B 0.000,C 90.000,E1 284.954} C_DIS
LIN {X -0.076,Y -445.201,Z 971.577,A 0.000,B 0.000,C 90.000,E1 283.883} C_DIS
LIN {X -0.017,Y -453.433,Z 971.571,A 0.000,B 0.000,C 90.000,E1 282.827} C_DIS
LIN {X 0.144,Y -461.244,Z 971.565,A 0.000,B 0.000,C 90.000,E1 281.771} C_DIS
LIN {X -0.149,Y -468.576,Z 971.560,A 0.000,B 0.000,C 90.000,E1 280.782} C_DIS
LIN {X -0.139,Y -473.662,Z 971.556,A 0.000,B 0.000,C 90.000,E1 280.018} C_DIS
LIN {X -0.164,Y -478.101,Z 971.551,A 0.000,B 0.000,C 90.000,E1 279.265} C_DIS
LIN {X -0.152,Y -481.896,Z 971.547,A 0.000,B 0.000,C 90.000,E1 278.511} C_DIS
LIN {X 0.013,Y -484.080,Z 971.544,A 0.000,B 0.000,C 90.000,E1 277.992} C_DIS
LIN {X 0.195,Y -485.964,Z 971.542,A 0.000,B 0.000,C 90.000,E1 277.473} C_DIS
LIN {X -0.039,Y -487.582,Z 971.539,A 0.000,B 0.000,C 90.000,E1 277.004} C_DIS
LIN {X 0.159,Y -488.862,Z 971.536,A 0.000,B 0.000,C 90.000,E1 276.486} C_DIS
LIN {X -0.121,Y -489.828,Z 971.533,A 0.000,B 0.000,C 90.000,E1 276.024} C_DIS
LIN {X 0.046,Y -490.417,Z 971.531,A 0.000,B 0.000,C 90.000,E1 275.511} C_DIS
LIN {X -0.219,Y -490.663,Z 971.528,A 0.000,B 0.000,C 90.000,E1 275.049} C_DIS
LIN {X 0.005,Y -490.521,Z 971.525,A 0.000,B 0.000,C 90.000,E1 274.531} C_DIS
LIN {X 0.228,Y -489.926,Z 971.522,A 0.000,B 0.000,C 90.000,E1 274.012} C_DIS
LIN {X -0.072,Y -488.819,Z 971.520,A 0.000,B 0.000,C 90.000,E1 273.555} C_DIS
LIN {X 0.142,Y -487.196,Z 971.517,A 0.000,B 0.000,C 90.000,E1 273.037} C_DIS
LIN {X -0.161,Y -484.898,Z 971.514,A 0.000,B 0.000,C 90.000,E1 272.579} C_DIS
LIN {X 0.008,Y -481.836,Z 971.511,A 0.000,B 0.000,C 90.000,E1 272.064} C_DIS
LIN {X -0.154,Y -480.058,Z 971.510,A 0.000,B 0.000,C 90.000,E1 271.835} C_DIS
LIN {X 0.176,Y -478.001,Z 971.509,A 0.000,B 0.000,C 90.000,E1 271.547} C_DIS
LIN {X -0.167,Y -473.132,Z 971.506,A 0.000,B 0.000,C 90.000,E1 271.088} C_DIS
LIN {X 0.039,Y -467.220,Z 971.503,A 0.000,B 0.000,C 90.000,E1 270.573} C_DIS
LIN {X -0.187,Y -460.995,Z 971.501,A 0.000,B 0.000,C 90.000,E1 270.172} C_DIS
LIN {X 0.031,Y -454.403,Z 971.499,A 0.000,B 0.000,C 90.000,E1 269.771} C_DIS
LIN {X -0.211,Y -447.546,Z 971.497,A 0.000,B 0.000,C 90.000,E1 269.484} C_DIS
LIN {X -0.056,Y -440.357,Z 971.495,A 0.000,B 0.000,C 90.000,E1 269.198} C_DIS
LIN {X 0.061,Y -432.961,Z 971.494,A 0.000,B 0.000,C 90.000,E1 268.969} C_DIS
LIN {X 0.068,Y -425.093,Z 971.493,A 0.000,B 0.000,C 90.000,E1 268.797} C_DIS
LIN {X -0.045,Y -417.293,Z 971.493,A 0.000,B 0.000,C 90.000,E1 268.682} C_DIS
